//Working Counter: Should remain Zero, If value=1 then data is bad from this device
g_xEP1908_Wc ;

*)

//END_IF ;

END_PROGRAM

// ---- POUs/Control_System_Diagnostics/System_Functions.TcPOU
PROGRAM System_Functions
//		8-2-2012
// 		This Program has been supplied by Beckhoff Automation As-Is and is intended only as an example 
//		implementation. Functionality is not guaranteed. 
//
VAR
	//General timer for periodic reads
	T1									:		TON ;
	xExecute							:		BOOL ;
	tTime1								:		TIME ;

	//Get Device Identification
	fbGetDeviceIdentificationEx			:		FB_GetDeviceIdentificationEx ;
	xGetDeviceId_Busy					:		BOOL ;
	xGetDeviceId_Error					:		BOOL ;
	udiGetDeviceId_ErrId				:		UDINT ;
	stDevIdent							:		ST_DeviceIdentificationEx ;

	//Get ADS Router Info
	fbGetRouterStatusInfo				:		FB_GetRouterStatusInfo ;
	xGetRouterStatusInfo_Busy			:		BOOL ;
	xGetRouterStatusInfo_Error			:		BOOL ;
	udiGetRouterStatusInfo_ErrId		:		UDINT ;
	stRouterStatusInfo					:		ST_TcRouterStatusInfo ;


(*
(* Get CPU Usage Info  *)
	fbTC_CpuUsage: TC_CpuUsage;
	bCpuUsage_Busy: BOOL;
	bCpuUsage_Error: BOOL;
	nCpuUsage_ErrId: UDINT;
	nCpuUsage: UDINT;
	nCpuUsage_HMI: UDINT;

(* Get System Latency Values *)
	fbTC_SysLatency: TC_SysLatency;
	bSysLatency_Busy: BOOL;
	bSysLatency_Error: BOOL;
	nSysLatency_ErrId: UDINT;
	nSysLatency_Actual: UDINT;
	nSysLatency_Max: UDINT;
	nSysLatency_Actual_HMI: UDINT;
	nSysLatency_Max_HMI: UDINT;

(* SystemTaskInfoArr[1].cycleTime is in 100ns increments - needed to convert to ms for display*)
	nCycleTime_HMI: LREAL;

(* SystemTaskInfoArr[1].lastExecTime is in 100ns increments - needed to convert to ms for display*)
	nLastExecTime_HMI: LREAL;
	fbGetDeviceIdentificationEx: FB_GetDeviceIdentificationEx;
*)
	fbFB_MDP_ScanModules				: 		FB_MDP_ScanModules;
	eMDP_ModType						: 		E_MDP_ModuleType;
	usiModIdx							: 		USINT;
	xMDP_ScanModules_busy				: 		BOOL;
	xMDP_ScanModules_Error				: 		BOOL;
	udiMDP_ScanModules_ErrID			: 		UDINT;
	bMDP_ScanModules_DynModID			: 		BYTE;
	usiMDP_ScanModules_ModTypCnt		: 		USINT;
	usiMDP_ScanModules_ModCnt			: 		USINT;

	fbFB_MDP_ReadModuleContent 			:		FB_MDP_ReadModuleContent ;
	ST_MDP_Addr 						:		ST_MDP_Addr ;
	dwMB_Buffer							: 		DWORD ;
	xMDP_Motherboard_ReadModContent_Busy: 		BOOL ;
	xMDP_Motherboard_ReadModContent_Error: 		BOOL ;
	udiMDP_Motherboard_ReadModContent_ErrID: 	UDINT ;
	usiMDP_Motherboard_ReadModContent_ErrPOS: 	USINT ;
	arrMDP_Motherboard_StartIdx			: 		ARRAY [0..255] OF UINT ;

	fbFB_MDP_SplitErrorID				: 		FB_MDP_SplitErrorID ;
	eMDP_ErrGroup 						:		E_MDP_ErrGroup ;
	uiMDP_Motherboard_ReadModContent_ErrCODE:	UINT ;

	fbFB_MDP_ReadModuleHeader			: 		FB_MDP_ReadModuleHeader ;
	xMDP_Motherboard_ReadModHeader_Busy	: 		BOOL ;
	xMDP_Motherboard_ReadModHeader_Error: 		BOOL ;
	udiMDP_Motherboard_ReadModHeader_ErrID: 	UDINT ;
	ST_MDP_Motherboard_ReadModHeader 	:		ST_MDP_ModuleHeader ;

	fbFB_MDP_CPU_Read1					: 		FB_MDP_CPU_Read;
	ST_CPUModHdr 						:		ST_MDP_ModuleHeader ;
	ST_CPUModContent 					: 		ST_MDP_CPU ;

	fbFB_MDP_Mainboard_ReadTBL1			: 		FB_MDP_Mainboard_ReadTBL1;
	ST_MainboardModHdrTBL1				:		ST_MDP_ModuleHeader ;
	ST_MainboardModContentTBL1			: 		ST_MDP_MainboardTBL1 ;

	fbFB_MDP_Mainboard_ReadTBL2			: 		FB_MDP_Mainboard_ReadTBL2 ;
	ST_MainboardModHdrTBL2				:		ST_MDP_ModuleHeader ;
	ST_MainboardModContentTBL2			: 		ST_MDP_MainboardTBL2 ;

	fbFB_MDP_Mainboard_ReadTBL3			: 		FB_MDP_Mainboard_ReadTBL3 ;
	ST_MainboardModHdrTBL3				:		ST_MDP_ModuleHeader ;
	ST_MainboardModContentTBL3			: 		ST_MDP_MainboardTBL3 ;

	fbFB_MDP_Mainboard_ReadTBL4			: 		FB_MDP_Mainboard_ReadTBL4 ;
	ST_MainboardModHdrTBL4				:		ST_MDP_ModuleHeader ;
	ST_MainboardModContentTBL4			: 		ST_MDP_MainboardTBL4 ;
	
	fbFB_MDP_NIC0_Read					: 		FB_MDP_NIC_Read ;
	ST_NIC0_ModHdr						: 		ST_MDP_ModuleHeader ;
	ST_NIC0_ModContent					: 		ST_MDP_NIC_Properties ;
	
	fbFB_MDP_NIC1_Read					: 		FB_MDP_NIC_Read ;
	ST_NIC1_ModHdr						: 		ST_MDP_ModuleHeader ;
	ST_NIC1_ModContent					: 		ST_MDP_NIC_Properties ;	
	lrOperTimeHrs						: 		LREAL ;
	lrOperTimeDays						: 		LREAL ;
	lrOperTimeYears						: 		LREAL ;

	fbFB_MDP_Time1_Read					: 		FB_MDP_Time_ReadTBL1 ;
	ST_Time1_ModHdr						: 		ST_MDP_ModuleHeader ;
	ST_Time1_ModContent					: 		ST_MDP_TimeTBL1 ;

	fbFB_MDP_Time2_Read					: 		FB_MDP_Time_ReadTBL2 ;
	ST_Time2_ModHdr						: 		ST_MDP_ModuleHeader ;
	ST_Time2_ModContent					: 		ST_MDP_TimeTBL2 ;
	
	fbFB_MDP_Memory_Read				: 		FB_MDP_Memory_ReadTBL1 ;
	ST_Memory_ModHdr					: 		ST_MDP_ModuleHeader ;
	ST_Memory_ModContent				: 		ST_MDP_MemoryTBL1 ;
	one									:		INT :=1 ;
	
//	fbFB_MDP_Time1_Read					: 		FB_MDP_Time_ReadTBL1 ;
//	ST_Memory_ModHdr					: 		ST_MDP_ModuleHeader ;
//	ST_Memory_ModContent				: 		ST_MDP_TimeTBL1 ;
	
	testword: INT;
	string45: STRING;
	fbFB_MDP_DiskMngmnt_ReadTBL1		: 		FB_MDP_DiskMngmnt_ReadTBL1 ;
	ST_DiskMngmnt_HdrTBL1				: 		ST_MDP_ModuleHeader ;
	ST_DiskMngmntTBL1					: 		ST_MDP_DiskMngmntTBL1 ;
END_VAR

//		8-2-2012
// 		This Program has been supplied by Beckhoff Automation As-Is and is intended only as an example 
//		implementation. Functionality is not guaranteed. 
//
//   ;
;
testword ;


//IF g_bHMI_ScreenBeingDisplayed = 90 THEN
//Create the xExecute bit for continuous timed interval FB calls
T1(IN:= NOT xExecute, PT:= T#2S, Q=> xExecute, ET=>tTime1 );

(* Computer/Controller Device Info - Get CX and TwinCAT version info
   from the resulting structure "stDevIdent" - display only when the 
   function block is not BUSY retrieving the data else the display
   will "blink" because while the FB is BUSY the values go to 0 or
   "blank" text *)
fbGetDeviceIdentificationEx(
							bExecute					:= 		xExecute, 
							tTimeout					:= 		T#2S, 
							sNetId						:= 		'', 
							bBusy						=> 		xGetDeviceId_Busy, 
							bError						=> 		xGetDeviceId_Error, 
							nErrorID					=> 		udiGetDeviceId_ErrId, 
							stDevIdent					=> 		stDevIdent );
							
IF NOT xGetDeviceId_Busy THEN 
							g_stHMI_DevIdent 			:= 		stDevIdent ; 
END_IF ;

g_stHMI_AppInfo 										:= _AppInfo  ;

//ADS Router Status info
fbGetRouterStatusInfo(		
							sNetId						:= 		'',
							bExecute					:= 		xExecute,
							tTimeout					:= 		T#2S,
							bBusy						=> 		xGetRouterStatusInfo_Busy,
							bError						=> 		xGetRouterStatusInfo_Error,
							nErrID						=> 		udiGetRouterStatusInfo_ErrId,
							info						=> 		stRouterStatusInfo );
							
IF NOT xGetRouterStatusInfo_Busy THEN 
							g_stHMI_RouterStatusInfo	:= 		stRouterStatusInfo ; 
END_IF ;

g_stHMI_PlcTaskSystemInfo 								:= 		_TaskInfo[_AppInfo.TaskCnt] ;
g_lrHMI_PlcTaskSystemInfo_CycleTime 					:= 		g_stHMI_PlcTaskSystemInfo.CycleTime / 10.0 ;
g_lrHMI_PlcTaskSystemInfo_LastExecTime 					:= 		g_stHMI_PlcTaskSystemInfo.LastExecTime / 10.0 ;

//In order to be able to query or set an MDP parameter, the Dynamic Module ID of 
//the module in which the parameter is located must be known.
fbFB_MDP_ScanModules(
							bExecute					:= 		xExecute, 
							nModuleType					:= 		eMDP_ModType, 
							iModIdx						:= 		usiModIdx, 
							tTimeout					:= 		T#2S, 
							sAmsNetId					:= 		'', 
							bBusy						=> 		xMDP_ScanModules_busy, 
							bError						=> 		xMDP_ScanModules_Error, 
							nErrID						=> 		udiMDP_ScanModules_ErrID, 
							nDynModuleId				=> 		bMDP_ScanModules_DynModID, 
							iModuleTypeCount			=> 		usiMDP_ScanModules_ModTypCnt, 
							iModuleCount				=> 		usiMDP_ScanModules_ModCnt );

// The function block enables the header of an MDP module to be queried
fbFB_MDP_ReadModuleHeader(
							bExecute					:= 		xExecute, 
							nDynModuleId				:= 		4, 
							tTimeout					:= 		T#2S, 
							sAmsNetId					:= 		'', 
							bBusy						=> 		xMDP_Motherboard_ReadModHeader_Busy, 
							bError						=> 		xMDP_Motherboard_ReadModHeader_Error, 
							nErrID						=> 		udiMDP_Motherboard_ReadModHeader_ErrID, 
							stMDP_ModHeader				=> 		ST_MDP_Motherboard_ReadModHeader);							
							

fbFB_MDP_CPU_Read1(
							xExecute					:= 		xExecute, 
							tTimeout					:= 		T#2S, 
							usiModIdx					:= 		0, 
							sAmsNetId					:= 		'', 
							bBusy						=> 		, 
							bError						=> 		, 
							nErrID						=> 		, 
							iErrPos						=> 		, 
							stMDP_ModuleHeader			=> 		ST_CPUModHdr, 
							stMDP_ModuleContent			=> 		ST_CPUModContent);							

g_lrHMI_CPUfrequency 									:=		ST_CPUModContent.udiCPUfrequency / 1000.0	; // CPU Clock Frequency in GHz				
g_iHMI_CPUusage											:=		ST_CPUModContent.uiCPUusage ;  // CPU Usage in percent
g_iHMI_CPUtemperature 									:= 		ST_CPUModContent.iCPUtemp ; // CPU Temperature in DegC	

fbFB_MDP_Mainboard_ReadTBL1(
							xExecute					:= 		xExecute, 
							tTimeout					:= 		T#2S, 
							usiModIdx					:= 		0, 
							sAmsNetId					:= 		'', 
							bBusy						=> 		, 
							bError						=> 		, 
							nErrID						=> 		, 
							iErrPos						=> 		, 
							stMDP_ModuleHeader			=> 		ST_MainboardModHdrTBL1, 
							stMDP_ModuleContent			=> 		ST_MainboardModContentTBL1);


g_sHMI_MainboardType 									:= 		ST_MainboardModContentTBL1.sMainboardType ;
g_sHMI_MainboardSN 										:= 		ST_MainboardModContentTBL1.sMainboardSN ;
g_sHMI_MainboardProdDate								:= 		ST_MainboardModContentTBL1.sMainboardProdDate ;
g_udiHMI_MainboardBootCount								:= 		ST_MainboardModContentTBL1.udiMainboardBootCount ;
lrOperTimeHrs											:= 		ST_MainboardModContentTBL1.udiMainboardOperTime / 60.0 ;
lrOperTimeDays											:= 		lrOperTimeHrs / 24.0 ;
g_udiHMI_MainboardOperTimeDays 							:= 		TRUNC(lrOperTimeDays) ;
g_lrHMI_MainboardOperTimeHrs							:=		24.0 * (lrOperTimeDays - UDINT_TO_LREAL(g_udiHMI_MainboardOperTimeDays)) ;
g_diHMI_MainboardMinTemp								:= 		ST_MainboardModContentTBL1.diMainboardMinTemp ;
g_diHMI_MainboardMaxTemp								:= 		ST_MainboardModContentTBL1.diMainboardMaxTemp ;
g_lrHMI_MainboardMinVolt								:= 		ST_MainboardModContentTBL1.diMainboardMinVolt / 1000.0 ;
g_lrHMI_MainboardMaxVolt								:= 		ST_MainboardModContentTBL1.diMainboardMaxVolt / 1000.0 ;
g_iHMI_MainboardActualTemp								:= 		ST_MainboardModContentTBL1.iMainboardActualTemp ;


fbFB_MDP_Mainboard_ReadTBL2(
							xExecute					:= 		xExecute, 
							tTimeout					:= 		T#2S, 
							usiModIdx						:= 		0, 
							sAmsNetId					:= 		'', 
							bBusy						=> 		, 
							bError						=> 		, 
							nErrID						=> 		, 
							iErrPos						=> 		, 
							stMDP_ModuleHeader			=> 		ST_MainboardModHdrTBL2, 
							stMDP_ModuleContent			=> 		ST_MainboardModContentTBL2);


g_bHMI_MainboardRevision 								:= 		ST_MainboardModContentTBL2.usiMainboardRevision ;
g_bHMI_MainboardBiosMajVers 							:= 		ST_MainboardModContentTBL2.usiMainboardBiosMajVers ;
g_bHMI_MainboardBiosMinVers 							:= 		ST_MainboardModContentTBL2.usiMainboardBiosMinVers ;


fbFB_MDP_Mainboard_ReadTBL3(
							xExecute					:= 		xExecute, 
							tTimeout					:= 		T#2S, 
							usiModIdx						:= 		0, 
							sAmsNetId					:= 		'', 
							bBusy						=> 		, 
							bError						=> 		, 
							nErrID						=> 		, 
							iErrPos						=> 		, 
							stMDP_ModuleHeader			=> 		ST_MainboardModHdrTBL3, 
							stMDP_ModuleContent			=> 		ST_MainboardModContentTBL3);							

g_sHMI_Mainboard1p05v 									:= 		ST_MainboardModContentTBL3.sMainboard1p05v ;
g_sHMI_MainboardVccCore 								:= 		ST_MainboardModContentTBL3.sMainboardVccCore ;
g_sHMI_Mainboard5v 										:= 		ST_MainboardModContentTBL3.sMainboard5v ;
g_sHMI_Mainboard12v 									:= 		ST_MainboardModContentTBL3.sMainboard12v ;
g_sHMI_MainboardVBatt 									:= 		ST_MainboardModContentTBL3.sMainboardVBatt ;
g_sHMI_MainboardPwrCtrlVcc 								:= 		ST_MainboardModContentTBL3.sMainboardPwrCtrlVcc ;
g_sHMI_MainboardCX2100_5v 								:= 		ST_MainboardModContentTBL3.sMainboardCX2100_5v ;
g_sHMI_MainboardCX2100_12v 								:= 		ST_MainboardModContentTBL3.sMainboardCX2100_12v ;
g_sHMI_MainboardCX2100_24v 								:= 		ST_MainboardModContentTBL3.sMainboardCX2100_24v ;

					
fbFB_MDP_Mainboard_ReadTBL4(
							xExecute					:= 		xExecute, 
							tTimeout					:= 		T#2S, 
							usiModIdx						:= 		0, 
							sAmsNetId					:= 		'', 
							bBusy						=> 		, 
							bError						=> 		, 
							nErrID						=> 		, 
							iErrPos						=> 		, 
							stMDP_ModuleHeader			=> 		ST_MainboardModHdrTBL4, 
							stMDP_ModuleContent			=> 		ST_MainboardModContentTBL4);

g_lrHMI_Mainboard1p05v 									:= 		ST_MainboardModContentTBL4.iMainboard1p05v / 1000.0 ;
g_lrHMI_MainboardVccCore 								:= 		ST_MainboardModContentTBL4.iMainboardVccCore / 1000.0 ;
g_lrHMI_Mainboard5v 									:= 		ST_MainboardModContentTBL4.iMainboard5v / 1000.0 ;
g_lrHMI_Mainboard12v 									:= 		ST_MainboardModContentTBL4.iMainboard12v / 1000.0 ;
g_lrHMI_MainboardVBatt 									:= 		ST_MainboardModContentTBL4.iMainboardVBatt / 1000.0 ;
g_lrHMI_MainboardPwrCtrlVcc 							:= 		ST_MainboardModContentTBL4.iMainboardPwrCtrlVcc / 1000.0 ;
g_lrHMI_MainboardCX2100_5v 								:= 		ST_MainboardModContentTBL4.iMainboardCX2100_5v / 1000.0 ;
g_lrHMI_MainboardCX2100_12v 							:= 		ST_MainboardModContentTBL4.iMainboardCX2100_12v / 1000.0 ;
g_lrHMI_MainboardCX2100_24v 							:= 		ST_MainboardModContentTBL4.iMainboardCX2100_24v / 1000.0 ; 


fbFB_MDP_NIC0_Read(
							xExecute					:= 		xExecute, 
							tTimeout					:= 		T#2S, 
							usiModIdx					:= 		0, 
							sAmsNetId					:= 		'', 
							bBusy						=> 		, 
							bError						=> 		, 
							nErrID						=> 		, 
							iErrPos						=> 		, 
							stMDP_ModuleHeader			=> 		ST_NIC0_ModHdr, 
							stMDP_ModuleContent			=> 		ST_NIC0_ModContent);

fbFB_MDP_NIC1_Read(
							xExecute					:= 		xExecute, 
							tTimeout					:= 		T#2S, 
							usiModIdx					:= 		1, 
							sAmsNetId					:= 		'', 
							bBusy						=> 		, 
							bError						=> 		, 
							nErrID						=> 		, 
							iErrPos						=> 		, 
							stMDP_ModuleHeader			=> 		ST_NIC1_ModHdr, 
							stMDP_ModuleContent			=> 		ST_NIC1_ModContent);

fbFB_MDP_Time1_Read(
							xExecute					:= 		xExecute, 
							tTimeout					:= 		T#2S, 
							usiModIdx					:= 		0, 
							sAmsNetId					:= 		'', 
							bBusy						=> 		, 
							bError						=> 		, 
							nErrID						=> 		, 
							iErrPos						=> 		, 
							stMDP_ModuleHeader			=> 		ST_Time1_ModHdr, 
							stMDP_ModuleContent			=> 		ST_Time1_ModContent);				

g_sHMI_SNTP_Server										:= 		ST_Time1_ModContent.sSNTP_Server ;
g_lrHMI_SNTP_Refresh_Minutes							:= 		UDINT_TO_LREAL(ST_Time1_ModContent.udiSNTP_Refresh) / 60.0 ; // Seconds / 60 = Minutes
g_lrHMI_Years_Since_1_1_1970							:= 		UDINT_TO_LREAL(ST_Time1_ModContent.udiSec_Since_1_1_1970) / (60 * 60 *24 * 365) ;
g_sHMI_DateTime_Presentation							:= 		ST_Time1_ModContent.sDateTime_Presentation ;
g_uiHMI_Timezone										:= 		ST_Time1_ModContent.uiTimezone ;


fbFB_MDP_Time2_Read(
							xExecute					:= 		xExecute, 
							tTimeout					:= 		T#2S, 
							usiModIdx					:= 		0, 
							sAmsNetId					:= 		'', 
							bBusy						=> 		, 
							bError						=> 		, 
							nErrID						=> 		, 
							iErrPos						=> 		, 
							stMDP_ModuleHeader			=> 		ST_Time2_ModHdr, 
							stMDP_ModuleContent			=> 		ST_Time2_ModContent);
							
IF ST_Time1_ModContent.uiTimezone = 0 THEN
	g_sHMI_currentTimeZone := ST_Time2_ModContent.sTimezone1 ;
ELSIF ST_Time1_ModContent.uiTimezone = 1 THEN
	g_sHMI_currentTimeZone := ST_Time2_ModContent.sTimezone2 ;
ELSIF ST_Time1_ModContent.uiTimezone = 2 THEN
	g_sHMI_currentTimeZone := ST_Time2_ModContent.sTimezone3 ;
ELSIF ST_Time1_ModContent.uiTimezone = 3 THEN
	g_sHMI_currentTimeZone := ST_Time2_ModContent.sTimezone4 ;
ELSIF ST_Time1_ModContent.uiTimezone = 4 THEN
	g_sHMI_currentTimeZone := ST_Time2_ModContent.sTimezone5 ;	
ELSIF ST_Time1_ModContent.uiTimezone = 5 THEN
	g_sHMI_currentTimeZone := ST_Time2_ModContent.sTimezone6 ;
ELSIF ST_Time1_ModContent.uiTimezone = 6 THEN
	g_sHMI_currentTimeZone := ST_Time2_ModContent.sTimezone7 ;
ELSIF ST_Time1_ModContent.uiTimezone = 7 THEN
	g_sHMI_currentTimeZone := ST_Time2_ModContent.sTimezone8 ;
ELSIF ST_Time1_ModContent.uiTimezone = 8 THEN
	g_sHMI_currentTimeZone := ST_Time2_ModContent.sTimezone9 ;		
ELSIF ST_Time1_ModContent.uiTimezone = 9 THEN
	g_sHMI_currentTimeZone := ST_Time2_ModContent.sTimezone10 ;
ELSIF ST_Time1_ModContent.uiTimezone = 10 THEN
	g_sHMI_currentTimeZone := ST_Time2_ModContent.sTimezone11 ;
ELSIF ST_Time1_ModContent.uiTimezone = 11 THEN
	g_sHMI_currentTimeZone := ST_Time2_ModContent.sTimezone12 ;
ELSIF ST_Time1_ModContent.uiTimezone = 12 THEN
	g_sHMI_currentTimeZone := ST_Time2_ModContent.sTimezone13 ;	
ELSIF ST_Time1_ModContent.uiTimezone = 13 THEN
	g_sHMI_currentTimeZone := ST_Time2_ModContent.sTimezone14 ;
ELSIF ST_Time1_ModContent.uiTimezone = 14 THEN
	g_sHMI_currentTimeZone := ST_Time2_ModContent.sTimezone15 ;
ELSIF ST_Time1_ModContent.uiTimezone = 15 THEN
	g_sHMI_currentTimeZone := ST_Time2_ModContent.sTimezone16 ;
ELSIF ST_Time1_ModContent.uiTimezone = 16 THEN
	g_sHMI_currentTimeZone := ST_Time2_ModContent.sTimezone17 ;		
ELSIF ST_Time1_ModContent.uiTimezone = 17 THEN
	g_sHMI_currentTimeZone := ST_Time2_ModContent.sTimezone18 ;
ELSIF ST_Time1_ModContent.uiTimezone = 18 THEN
	g_sHMI_currentTimeZone := ST_Time2_ModContent.sTimezone19 ;
ELSIF ST_Time1_ModContent.uiTimezone = 19 THEN
	g_sHMI_currentTimeZone := ST_Time2_ModContent.sTimezone20 ;
ELSIF ST_Time1_ModContent.uiTimezone = 20 THEN
	g_sHMI_currentTimeZone := ST_Time2_ModContent.sTimezone21 ;	
ELSIF ST_Time1_ModContent.uiTimezone = 21 THEN
	g_sHMI_currentTimeZone := ST_Time2_ModContent.sTimezone22 ;
ELSIF ST_Time1_ModContent.uiTimezone = 22 THEN
	g_sHMI_currentTimeZone := ST_Time2_ModContent.sTimezone23 ;
ELSIF ST_Time1_ModContent.uiTimezone = 23 THEN
	g_sHMI_currentTimeZone := ST_Time2_ModContent.sTimezone24 ;
ELSIF ST_Time1_ModContent.uiTimezone = 24 THEN
	g_sHMI_currentTimeZone := ST_Time2_ModContent.sTimezone25 ;		
ELSIF ST_Time1_ModContent.uiTimezone = 25 THEN
	g_sHMI_currentTimeZone := ST_Time2_ModContent.sTimezone26 ;
ELSIF ST_Time1_ModContent.uiTimezone = 26 THEN
	g_sHMI_currentTimeZone := ST_Time2_ModContent.sTimezone27 ;
ELSIF ST_Time1_ModContent.uiTimezone = 27 THEN
	g_sHMI_currentTimeZone := ST_Time2_ModContent.sTimezone28 ;
ELSIF ST_Time1_ModContent.uiTimezone = 28 THEN
	g_sHMI_currentTimeZone := ST_Time2_ModContent.sTimezone29 ;	
ELSIF ST_Time1_ModContent.uiTimezone = 29 THEN
	g_sHMI_currentTimeZone := ST_Time2_ModContent.sTimezone30 ;
ELSIF ST_Time1_ModContent.uiTimezone = 30 THEN
	g_sHMI_currentTimeZone := ST_Time2_ModContent.sTimezone31 ;
ELSIF ST_Time1_ModContent.uiTimezone = 31 THEN
	g_sHMI_currentTimeZone := ST_Time2_ModContent.sTimezone32 ;
ELSIF ST_Time1_ModContent.uiTimezone = 32 THEN
	g_sHMI_currentTimeZone := ST_Time2_ModContent.sTimezone33 ;			
ELSIF ST_Time1_ModContent.uiTimezone = 33 THEN
	g_sHMI_currentTimeZone := ST_Time2_ModContent.sTimezone34 ;
ELSIF ST_Time1_ModContent.uiTimezone = 34 THEN
	g_sHMI_currentTimeZone := ST_Time2_ModContent.sTimezone35 ;
ELSIF ST_Time1_ModContent.uiTimezone = 35 THEN
	g_sHMI_currentTimeZone := ST_Time2_ModContent.sTimezone36 ;
ELSIF ST_Time1_ModContent.uiTimezone = 36 THEN
	g_sHMI_currentTimeZone := ST_Time2_ModContent.sTimezone37 ;	
ELSIF ST_Time1_ModContent.uiTimezone = 37 THEN
	g_sHMI_currentTimeZone := ST_Time2_ModContent.sTimezone38 ;
ELSIF ST_Time1_ModContent.uiTimezone = 38 THEN
	g_sHMI_currentTimeZone := ST_Time2_ModContent.sTimezone39 ;
ELSIF ST_Time1_ModContent.uiTimezone = 39 THEN
	g_sHMI_currentTimeZone := ST_Time2_ModContent.sTimezone40 ;
ELSIF ST_Time1_ModContent.uiTimezone = 40 THEN
	g_sHMI_currentTimeZone := ST_Time2_ModContent.sTimezone41 ;		
ELSIF ST_Time1_ModContent.uiTimezone = 41 THEN
	g_sHMI_currentTimeZone := ST_Time2_ModContent.sTimezone42 ;
ELSIF ST_Time1_ModContent.uiTimezone = 42 THEN
	g_sHMI_currentTimeZone := ST_Time2_ModContent.sTimezone43 ;
ELSIF ST_Time1_ModContent.uiTimezone = 43 THEN
	g_sHMI_currentTimeZone := ST_Time2_ModContent.sTimezone44 ;
ELSIF ST_Time1_ModContent.uiTimezone = 44 THEN
	g_sHMI_currentTimeZone := ST_Time2_ModContent.sTimezone45 ;	
ELSIF ST_Time1_ModContent.uiTimezone = 45 THEN
	g_sHMI_currentTimeZone := ST_Time2_ModContent.sTimezone46 ;
ELSIF ST_Time1_ModContent.uiTimezone = 46 THEN
	g_sHMI_currentTimeZone := ST_Time2_ModContent.sTimezone47 ;
ELSIF ST_Time1_ModContent.uiTimezone = 47 THEN
	g_sHMI_currentTimeZone := ST_Time2_ModContent.sTimezone48 ;
ELSIF ST_Time1_ModContent.uiTimezone = 48 THEN
	g_sHMI_currentTimeZone := ST_Time2_ModContent.sTimezone49 ;		
ELSIF ST_Time1_ModContent.uiTimezone = 49 THEN
	g_sHMI_currentTimeZone := ST_Time2_ModContent.sTimezone50 ;
ELSIF ST_Time1_ModContent.uiTimezone = 50 THEN
	g_sHMI_currentTimeZone := ST_Time2_ModContent.sTimezone51 ;
ELSIF ST_Time1_ModContent.uiTimezone = 51 THEN
	g_sHMI_currentTimeZone := ST_Time2_ModContent.sTimezone52 ;
ELSIF ST_Time1_ModContent.uiTimezone = 52 THEN
	g_sHMI_currentTimeZone := ST_Time2_ModContent.sTimezone53 ;	
ELSIF ST_Time1_ModContent.uiTimezone = 53 THEN
	g_sHMI_currentTimeZone := ST_Time2_ModContent.sTimezone54 ;
ELSIF ST_Time1_ModContent.uiTimezone = 54 THEN
	g_sHMI_currentTimeZone := ST_Time2_ModContent.sTimezone55 ;
ELSIF ST_Time1_ModContent.uiTimezone = 55 THEN
	g_sHMI_currentTimeZone := ST_Time2_ModContent.sTimezone56 ;
ELSIF ST_Time1_ModContent.uiTimezone = 56 THEN
	g_sHMI_currentTimeZone := ST_Time2_ModContent.sTimezone57 ;		
ELSIF ST_Time1_ModContent.uiTimezone = 57 THEN
	g_sHMI_currentTimeZone := ST_Time2_ModContent.sTimezone58 ;
ELSIF ST_Time1_ModContent.uiTimezone = 58 THEN
	g_sHMI_currentTimeZone := ST_Time2_ModContent.sTimezone59 ;
ELSIF ST_Time1_ModContent.uiTimezone = 59 THEN
	g_sHMI_currentTimeZone := ST_Time2_ModContent.sTimezone60 ;
ELSIF ST_Time1_ModContent.uiTimezone = 60 THEN
	g_sHMI_currentTimeZone := ST_Time2_ModContent.sTimezone61 ;	
ELSIF ST_Time1_ModContent.uiTimezone = 61 THEN
	g_sHMI_currentTimeZone := ST_Time2_ModContent.sTimezone62 ;
ELSIF ST_Time1_ModContent.uiTimezone = 62 THEN
	g_sHMI_currentTimeZone := ST_Time2_ModContent.sTimezone63 ;
ELSIF ST_Time1_ModContent.uiTimezone = 63 THEN
	g_sHMI_currentTimeZone := ST_Time2_ModContent.sTimezone64 ;
ELSIF ST_Time1_ModContent.uiTimezone = 64 THEN
	g_sHMI_currentTimeZone := ST_Time2_ModContent.sTimezone65 ;	
ELSIF ST_Time1_ModContent.uiTimezone = 65 THEN
	g_sHMI_currentTimeZone := ST_Time2_ModContent.sTimezone66 ;
ELSIF ST_Time1_ModContent.uiTimezone = 66 THEN
	g_sHMI_currentTimeZone := ST_Time2_ModContent.sTimezone67 ;
ELSIF ST_Time1_ModContent.uiTimezone = 67 THEN
	g_sHMI_currentTimeZone := ST_Time2_ModContent.sTimezone68 ;
ELSIF ST_Time1_ModContent.uiTimezone = 68 THEN
	g_sHMI_currentTimeZone := ST_Time2_ModContent.sTimezone69 ;	
ELSIF ST_Time1_ModContent.uiTimezone = 69 THEN
	g_sHMI_currentTimeZone := ST_Time2_ModContent.sTimezone70 ;
ELSIF ST_Time1_ModContent.uiTimezone = 70 THEN
	g_sHMI_currentTimeZone := ST_Time2_ModContent.sTimezone71 ;
ELSIF ST_Time1_ModContent.uiTimezone = 71 THEN
	g_sHMI_currentTimeZone := ST_Time2_ModContent.sTimezone72 ;
ELSIF ST_Time1_ModContent.uiTimezone = 72 THEN
	g_sHMI_currentTimeZone := ST_Time2_ModContent.sTimezone73 ;		
ELSIF ST_Time1_ModContent.uiTimezone = 73 THEN
	g_sHMI_currentTimeZone := ST_Time2_ModContent.sTimezone74 ;
ELSIF ST_Time1_ModContent.uiTimezone = 74 THEN
	g_sHMI_currentTimeZone := ST_Time2_ModContent.sTimezone75 ;
ELSIF ST_Time1_ModContent.uiTimezone = 75 THEN
	g_sHMI_currentTimeZone := ST_Time2_ModContent.sTimezone76 ;
ELSIF ST_Time1_ModContent.uiTimezone = 76 THEN
	g_sHMI_currentTimeZone := ST_Time2_ModContent.sTimezone77 ;	
ELSIF ST_Time1_ModContent.uiTimezone = 77 THEN
	g_sHMI_currentTimeZone := ST_Time2_ModContent.sTimezone78 ;
ELSIF ST_Time1_ModContent.uiTimezone = 78 THEN
	g_sHMI_currentTimeZone := ST_Time2_ModContent.sTimezone79 ;
ELSIF ST_Time1_ModContent.uiTimezone = 79 THEN
	g_sHMI_currentTimeZone := ST_Time2_ModContent.sTimezone80 ;
ELSIF ST_Time1_ModContent.uiTimezone = 80 THEN
	g_sHMI_currentTimeZone := ST_Time2_ModContent.sTimezone81 ;		
ELSIF ST_Time1_ModContent.uiTimezone = 81 THEN
	g_sHMI_currentTimeZone := ST_Time2_ModContent.sTimezone82 ;
ELSIF ST_Time1_ModContent.uiTimezone = 82 THEN
	g_sHMI_currentTimeZone := ST_Time2_ModContent.sTimezone83 ;
ELSIF ST_Time1_ModContent.uiTimezone = 83 THEN
	g_sHMI_currentTimeZone := ST_Time2_ModContent.sTimezone84 ;
ELSIF ST_Time1_ModContent.uiTimezone = 84 THEN
	g_sHMI_currentTimeZone := ST_Time2_ModContent.sTimezone85 ;	
ELSIF ST_Time1_ModContent.uiTimezone = 85 THEN
	g_sHMI_currentTimeZone := ST_Time2_ModContent.sTimezone86 ;
ELSIF ST_Time1_ModContent.uiTimezone = 86 THEN
	g_sHMI_currentTimeZone := ST_Time2_ModContent.sTimezone87 ;
ELSIF ST_Time1_ModContent.uiTimezone = 87 THEN
	g_sHMI_currentTimeZone := ST_Time2_ModContent.sTimezone88 ;
ELSIF ST_Time1_ModContent.uiTimezone = 88 THEN
	g_sHMI_currentTimeZone := ST_Time2_ModContent.sTimezone89 ;		
ELSIF ST_Time1_ModContent.uiTimezone = 89 THEN
	g_sHMI_currentTimeZone := ST_Time2_ModContent.sTimezone90 ;
ELSIF ST_Time1_ModContent.uiTimezone = 90 THEN
	g_sHMI_currentTimeZone := ST_Time2_ModContent.sTimezone91 ;
ELSIF ST_Time1_ModContent.uiTimezone = 91 THEN
	g_sHMI_currentTimeZone := ST_Time2_ModContent.sTimezone92 ;
ELSIF ST_Time1_ModContent.uiTimezone = 92 THEN
	g_sHMI_currentTimeZone := ST_Time2_ModContent.sTimezone93 ;	
ELSIF ST_Time1_ModContent.uiTimezone = 93 THEN
	g_sHMI_currentTimeZone := ST_Time2_ModContent.sTimezone94 ;
ELSIF ST_Time1_ModContent.uiTimezone = 94 THEN
	g_sHMI_currentTimeZone := ST_Time2_ModContent.sTimezone95 ;
ELSIF ST_Time1_ModContent.uiTimezone = 95 THEN
	g_sHMI_currentTimeZone := ST_Time2_ModContent.sTimezone96 ;
ELSIF ST_Time1_ModContent.uiTimezone = 96 THEN
	g_sHMI_currentTimeZone := ST_Time2_ModContent.sTimezone97 ;			
ELSIF ST_Time1_ModContent.uiTimezone = 97 THEN
	g_sHMI_currentTimeZone := ST_Time2_ModContent.sTimezone98 ;
ELSIF ST_Time1_ModContent.uiTimezone = 98 THEN
	g_sHMI_currentTimeZone := ST_Time2_ModContent.sTimezone99 ;
ELSIF ST_Time1_ModContent.uiTimezone = 99 THEN
	g_sHMI_currentTimeZone := ST_Time2_ModContent.sTimezone100 ;
ELSIF ST_Time1_ModContent.uiTimezone = 100 THEN
	g_sHMI_currentTimeZone := ST_Time2_ModContent.sTimezone101 ;	
END_IF
							
fbFB_MDP_Memory_Read(
							xExecute					:= 		xExecute, 
							tTimeout					:= 		T#2S, 
							usiModIdx					:= 		0, 
							sAmsNetId					:= 		'', 
							bBusy						=> 		, 
							bError						=> 		, 
							nErrID						=> 		, 
							iErrPos						=> 		, 
							stMDP_ModuleHeader			=> 		ST_Memory_ModHdr, 
							stMDP_ModuleContent			=> 		ST_Memory_ModContent);		

	g_lrHMI_ProgMemAllocated_InGB 		:= UDINT_TO_LREAL(ST_Memory_ModContent.udiProgMemAllocated) / 1000000000.0 ;	
	g_lrHMI_ProgMemAvailable_InGB 		:= UDINT_TO_LREAL(ST_Memory_ModContent.udiProgMemAvailable) / 1000000000.0 ;	
	g_lrHMI_ProgMemUsed_InGB 			:= g_lrHMI_ProgMemAllocated_InGB - g_lrHMI_ProgMemAvailable_InGB ;	
	g_lrHMI_ProgStorAllocated_InGB 		:= UDINT_TO_LREAL(ST_Memory_ModContent.udiStorageMemAllocated) / 1000000000.0 ;	
	g_lrHMI_ProgStorAvailable_InGB 		:= UDINT_TO_LREAL(ST_Memory_ModContent.udiStorageMemAvailable) / 1000000000.0 ;	
	g_lrHMI_ProgStorUsed_InGB 			:= g_lrHMI_ProgStorAllocated_InGB - g_lrHMI_ProgStorAvailable_InGB ;
	g_lrHMI_ProgStorMemDivision_InGB	:= UDINT_TO_LREAL(ST_Memory_ModContent.udiMemoryDivision) / 1000000000.0 ;	


fbFB_MDP_DiskMngmnt_ReadTBL1(
								xExecute				:= 		xExecute, 
								tTimeout				:= 		T#2S, 
								usiModIdx				:= 		0, 
								sAmsNetId				:= 		'', 
								bBusy					=> 		, 
								bError					=> 		, 
								nErrID					=> 		, 
								iErrPos					=> 		, 
								stMDP_ModuleHeader		=> 		ST_DiskMngmnt_HdrTBL1, 
								stMDP_ModuleContent		=> 		ST_DiskMngmntTBL1);








							
fbFB_MDP_Time1_Read(
							xExecute					:= 		xExecute, 
							tTimeout					:= 		T#2S, 
							usiModIdx					:= 		0, 
							sAmsNetId					:= 		'', 
							bBusy						=> 		, 
							bError						=> 		, 
							nErrID						=> 		, 
							iErrPos						=> 		, 
							stMDP_ModuleHeader			=> 		ST_Time1_ModHdr, 
							stMDP_ModuleContent			=> 		ST_Time1_ModContent);					
//	END_IF ;

END_PROGRAM

// ---- POUs/MDP_Function_Blocks/FB_MDP_CPU_Read.TcPOU
FUNCTION_BLOCK FB_MDP_CPU_Read

VAR_INPUT
	xExecute			: BOOL;								// Function block execution is triggered by a rising edge at this input
	tTimeout			: TIME		:= DEFAULT_ADS_TIMEOUT;	// States the time before the function is cancelled
	usiModIdx			: USINT		:= 0;					// Index number of chosen MDP device
	sAmsNetId			: T_AmsNetId;						// keep empty '' for the local device
END_VAR

VAR_OUTPUT
	xBusy				: BOOL;
	xError				: BOOL;
	udiErrID			: UDINT;
	usiErrPos			: USINT;							//If a subindex is not supported, iErrPos indicates at which subindex the error appears first
	stMDP_ModuleHeader	: ST_MDP_ModuleHeader;
	stMDP_ModuleContent	: ST_MDP_CPU;	
END_VAR

VAR
	fbMDP_ReadModule: FB_MDP_ReadModule;
	arrData				: ARRAY[0..15] OF BYTE;				// requested data
	arrStartIdx			: ARRAY[0..255] OF UINT;			// startindexes in bytes of each subindex element

	stMDP_Addr			: ST_MDP_Addr;
	eModuleType			: E_MDP_ModuleType;
	usiSubIdxCount		: USINT;

	xSubExecute			: BOOL;
	xReadBusy			: BOOL;

	RisingEdge			: R_TRIG;
	TimeOut				: TON;								// general timeout	
END_VAR

RisingEdge( CLK					:= xExecute );
IF NOT xBusy THEN											// FB only react to the external execute if it is not busy
	IF RisingEdge.Q THEN
		xBusy					:= TRUE;

		// reset variables
		xError					:= FALSE;
		udiErrID				:= 0;
		usiErrPos				:= 0;
		xSubExecute				:= TRUE;

		// specific values for CPU content
		stMDP_Addr.nArea		:= 16#08;
//		stMDP_Addr.nModuleId;								will be allocated dynamically
		stMDP_Addr.nTableId		:= 16#01;
//		stMDP_Addr.nFlag;									not used at ths time
//		stMDP_Addr.nSubIdx;									all subindexes will be requested
		eModuleType				:= eMDP_ModT_CPU;
		usiSubIdxCount			:= 4;						// TableId 16#01 contains 3 elements

		MEMSET( ADR(arrData), 0, SIZEOF(arrData) );			// reset buffer

		TimeOut(IN 				:= FALSE);
		TimeOut(PT 				:= tTimeout, IN 	:= TRUE);
	END_IF
END_IF


IF xBusy THEN
	IF xSubExecute THEN
		xSubExecute 			:= FALSE;

		fbMDP_ReadModule( bExecute := FALSE );
		fbMDP_ReadModule(
			stMDP_Addr			:= stMDP_Addr,
			eModuleType			:= eModuleType,
			iModIdx				:= usiModIdx,
			iSubIdxCount		:= usiSubIdxCount,
			bExecute			:= TRUE,
			tTimeout			:= tTimeout,
			pDstBuf				:= ADR(arrData),
			cbDstBufLen			:= SIZEOF(arrData),
			sAmsNetId			:= sAmsNetId,

			bBusy				=> xReadBusy,
			bError				=> xError,
			nErrID				=> udiErrID,
			iErrPos				=> usiErrPos,
			stMDP_DynAddr		=> ,
			iModuleTypeCount	=> ,
			iModuleCount		=> ,
			stMDP_ModuleHeader	=> ,
			arrStartIdx			=> ,
		);
	ELSE
		fbMDP_ReadModule(
			bExecute			:= FALSE,

			bBusy				=> xReadBusy,
			bError				=> xError,
			nErrID 				=> udiErrID,
			iErrPos				=> usiErrPos,
		 );
		IF NOT xReadBusy THEN
			// allocate received module header
			stMDP_ModuleHeader	:= fbMDP_ReadModule.stMDP_ModuleHeader;
			// allocate information of startindexes in data buffer
			MEMCPY(ADR(arrStartIdx), ADR(fbMDP_ReadModule.arrStartIdx), SIZEOF(arrStartIdx) );
			// reset module content struct
			MEMSET( ADR(stMDP_ModuleContent), 0, SIZEOF(stMDP_ModuleContent) );
			// allocate received data to NIC struct
			stMDP_ModuleContent.uiLen		:= arrData[0];
			MEMCPY(ADR(stMDP_ModuleContent.udiCPUfrequency), 	ADR(arrData)+arrStartIdx[1], MIN(arrStartIdx[2]-arrStartIdx[1], SIZEOF(stMDP_ModuleContent.udiCPUfrequency)) );
			MEMCPY(ADR(stMDP_ModuleContent.uiCPUusage), 		ADR(arrData)+arrStartIdx[2], MIN(arrStartIdx[3]-arrStartIdx[2], SIZEOF(stMDP_ModuleContent.uiCPUusage))     );
			MEMCPY(ADR(stMDP_ModuleContent.iCPUtemp), 			ADR(arrData)+arrStartIdx[3], MIN(arrStartIdx[4]-arrStartIdx[3], SIZEOF(stMDP_ModuleContent.iCPUtemp))     );

			// reset FB
			xBusy 				:= FALSE;
		END_IF
	END_IF

	
	// check timeout
	TimeOut();
	IF TimeOut.Q THEN
		TimeOut(IN 				:= FALSE);
		xError					:= TRUE;
		udiErrID				:= INT_TO_UINT(eMDP_Err_PLC) * 16#10000 + INT_TO_UINT(eMDP_ErrPLC_TimeOut);
	END_IF
END_IF

IF xError THEN
	// reset FB
	xBusy := FALSE;
END_IF

END_FUNCTION_BLOCK

// ---- POUs/MDP_Function_Blocks/FB_MDP_Mainboard_ReadTBL2.TcPOU
FUNCTION_BLOCK FB_MDP_Mainboard_ReadTBL2

VAR_INPUT
	xExecute			: BOOL;								// Function block execution is triggered by a rising edge at this input
	tTimeout			: TIME		:= DEFAULT_ADS_TIMEOUT;	// States the time before the function is cancelled
	usiModIdx			: USINT		:= 0;					// Index number of chosen MDP device 
	sAmsNetId			: T_AmsNetId;						// keep empty '' for the local device
END_VAR

VAR_OUTPUT
	xBusy				: BOOL;
	xError				: BOOL;
	udiErrID			: UDINT;
	usiErrPos			: USINT;							// If a subindex is not supported, iErrPos indicates at which subindex the error appears first
	stMDP_ModuleHeader	: ST_MDP_ModuleHeader;
	stMDP_ModuleContent	: ST_MDP_MainboardTBL2;	
END_VAR

VAR
	fbMDP_ReadModule: FB_MDP_ReadModule;
	arrData				: ARRAY[0..5] OF BYTE;				// requested data
	arrStartIdx			: ARRAY[0..4] OF UINT;				// startindexes in bytes of each subindex element

	stMDP_Addr			: ST_MDP_Addr;
	eModuleType			: E_MDP_ModuleType;
	usiSubIdxCount		: USINT;

	xSubExecute			: BOOL;
	xReadBusy			: BOOL;

	RisingEdge			: R_TRIG;
	TimeOut				: TON;								// general timeout	
END_VAR

RisingEdge( CLK					:= xExecute );
IF NOT xBusy THEN										// FB only react to the external execute if it is not busy
	IF RisingEdge.Q THEN
		xBusy					:= TRUE;
		// reset variables
		xError					:= FALSE;
		udiErrID				:= 0;
		usiErrPos				:= 0;
		xSubExecute				:= TRUE;

		// specific values for Mainboard content
		stMDP_Addr.nArea		:= 16#08;
//		stMDP_Addr.nModuleId;							will be allocated dynamically
		stMDP_Addr.nTableId		:= 16#02;
//		stMDP_Addr.nFlag;								not used up to now
//		stMDP_Addr.nSubIdx;								all subindexes will be requested
		eModuleType				:= eMDP_ModT_Mainboard;
		usiSubIdxCount			:= 4;					// TableId 16#01 contains 3 elements

		MEMSET( ADR(arrData), 0, SIZEOF(arrData) );		// reset buffer

		TimeOut(IN 				:= FALSE);
		TimeOut(PT 				:= tTimeout, IN 	:= TRUE);
	END_IF
END_IF


IF xBusy THEN
	IF xSubExecute THEN
		xSubExecute 			:= FALSE;

		fbMDP_ReadModule( bExecute := FALSE );
		fbMDP_ReadModule(
			stMDP_Addr			:= stMDP_Addr,
			eModuleType			:= eModuleType,
			iModIdx				:= usiModIdx,
			iSubIdxCount		:= usiSubIdxCount,
			bExecute			:= TRUE,
			tTimeout			:= tTimeout,
			pDstBuf				:= ADR(arrData),
			cbDstBufLen			:= SIZEOF(arrData),
			sAmsNetId			:= sAmsNetId,

			bBusy				=> xReadBusy,
			bError				=> xError,
			nErrID				=> udiErrID,
			iErrPos				=> usiErrPos,
			stMDP_DynAddr		=> ,
			iModuleTypeCount	=> ,
			iModuleCount		=> ,
			stMDP_ModuleHeader	=> ,
			arrStartIdx			=> ,
		);
	ELSE
		fbMDP_ReadModule(
			bExecute			:= FALSE,

			bBusy				=> xReadBusy,
			bError				=> xError,
			nErrID 				=> udiErrID,
			iErrPos				=> usiErrPos,
		 );
		IF NOT xReadBusy THEN
			// allocate received module header
			stMDP_ModuleHeader	:= fbMDP_ReadModule.stMDP_ModuleHeader;
			// allocate information of startindexes in data buffer
			MEMCPY(ADR(arrStartIdx), ADR(fbMDP_ReadModule.arrStartIdx), SIZEOF(arrStartIdx) );
			// reset module content struct
			MEMSET( ADR(stMDP_ModuleContent), 0, SIZEOF(stMDP_ModuleContent) );
			// allocate received data to NIC struct
			stMDP_ModuleContent.uiLen		:= arrData[0];
			MEMCPY(ADR(stMDP_ModuleContent.usiMainboardRevision),			ADR(arrData)+arrStartIdx[1],	MIN(arrStartIdx[2]-arrStartIdx[1],	SIZEOF(stMDP_ModuleContent.usiMainboardRevision))     );
			MEMCPY(ADR(stMDP_ModuleContent.usiMainboardBiosMajVers),		ADR(arrData)+arrStartIdx[2],	MIN(arrStartIdx[3]-arrStartIdx[2],	SIZEOF(stMDP_ModuleContent.usiMainboardBiosMajVers))     );
			MEMCPY(ADR(stMDP_ModuleContent.usiMainboardBiosMinVers),		ADR(arrData)+arrStartIdx[3],	MIN(arrStartIdx[4]-arrStartIdx[3],	SIZEOF(stMDP_ModuleContent.usiMainboardBiosMinVers))     );

			// reset FB
			xBusy 				:= FALSE;
		END_IF
	END_IF

	// check timeout
	TimeOut();
	IF TimeOut.Q THEN
		TimeOut(IN 				:= FALSE);
		xError					:= TRUE;
		udiErrID				:= INT_TO_UINT(eMDP_Err_PLC) * 16#10000 + INT_TO_UINT(eMDP_ErrPLC_TimeOut);
	END_IF
END_IF

IF xError THEN
	// reset FB
	xBusy 						:= FALSE;
END_IF

END_FUNCTION_BLOCK

// ---- POUs/MDP_Function_Blocks/FB_MDP_Mainboard_ReadTBL3.TcPOU
FUNCTION_BLOCK FB_MDP_Mainboard_ReadTBL3

VAR_INPUT
	xExecute				: BOOL;								// Function block execution is triggered by a rising edge at this input
	tTimeout				: TIME		:= DEFAULT_ADS_TIMEOUT;	// States the time before the function is cancelled
	usiModIdx				: USINT		:= 0;					// Index number of chosen MDP device
	sAmsNetId				: T_AmsNetId;						// keep empty '' for the local device
END_VAR

VAR_OUTPUT
	xBusy					: BOOL;
	xError					: BOOL;
	udiErrID				: UDINT;
	usiErrPos				: USINT;							// If a subindex is not supported, iErrPos indicates at which subindex the error appears first
	stMDP_ModuleHeader		: ST_MDP_ModuleHeader;
	stMDP_ModuleContent		: ST_MDP_MainboardTBL3;	
END_VAR

VAR
	fbMDP_ReadModule		: FB_MDP_ReadModule;
	arrData					: ARRAY[0..70] OF BYTE;				// requested data
	arrStartIdx				: ARRAY[0..11] OF UINT;				// startindexes in bytes of each subindex element

	stMDP_Addr				: ST_MDP_Addr;
	eModuleType				: E_MDP_ModuleType;
	usiSubIdxCount			: USINT;

	xSubExecute				: BOOL;
	xReadBusy				: BOOL;

	RisingEdge				: R_TRIG;
	TimeOut					: TON;								// general timeout	
END_VAR

RisingEdge( CLK					:= xExecute );
IF NOT xBusy THEN											// FB only react to the external execute if it is not busy
	IF RisingEdge.Q THEN
		xBusy					:= TRUE;

		// reset variables
		xError					:= FALSE;
		udiErrID				:= 0;
		usiErrPos				:= 0;
		xSubExecute				:= TRUE;

		// specific values for Mainboard content
		stMDP_Addr.nArea		:= 16#08;
//		stMDP_Addr.nModuleId;								will be allocated dynamically
		stMDP_Addr.nTableId		:= 16#03;
//		stMDP_Addr.nFlag;									not used at this time
//		stMDP_Addr.nSubIdx;									all subindexes will be requested
		eModuleType				:= eMDP_ModT_Mainboard;
		usiSubIdxCount			:= 10;						// TableId 16#01 contains 9 elements

		MEMSET( ADR(arrData), 0, SIZEOF(arrData) );			// reset buffer

		TimeOut(IN 				:= FALSE);
		TimeOut(PT 				:= tTimeout, IN 	:= TRUE);
	END_IF
END_IF


IF xBusy THEN
	IF xSubExecute THEN
		xSubExecute 			:= FALSE;

		fbMDP_ReadModule( bExecute := FALSE );
		fbMDP_ReadModule(
			stMDP_Addr			:= stMDP_Addr,
			eModuleType			:= eModuleType,
			iModIdx				:= usiModIdx,
			iSubIdxCount		:= usiSubIdxCount,
			bExecute			:= TRUE,
			tTimeout			:= tTimeout,
			pDstBuf				:= ADR(arrData),
			cbDstBufLen			:= SIZEOF(arrData),
			sAmsNetId			:= sAmsNetId,

			bBusy				=> xReadBusy,
			bError				=> xError,
			nErrID				=> udiErrID,
			iErrPos				=> usiErrPos,
			stMDP_DynAddr		=> ,
			iModuleTypeCount	=> ,
			iModuleCount		=> ,
			stMDP_ModuleHeader	=> ,
			arrStartIdx			=> ,
		);
	ELSE
		fbMDP_ReadModule(
			bExecute			:= FALSE,

			bBusy				=> xReadBusy,
			bError				=> xError,
			nErrID 				=> udiErrID,
			iErrPos				=> usiErrPos,
		 );
		IF NOT xReadBusy THEN
			// allocate received module header
			stMDP_ModuleHeader	:= fbMDP_ReadModule.stMDP_ModuleHeader;
			// allocate information of startindexes in data buffer
			MEMCPY(ADR(arrStartIdx), ADR(fbMDP_ReadModule.arrStartIdx), SIZEOF(arrStartIdx) );
			// reset module content struct
			MEMSET( ADR(stMDP_ModuleContent), 0, SIZEOF(stMDP_ModuleContent) );
			// allocate received data to NIC struct
			stMDP_ModuleContent.uiLen		:= arrData[0];
			MEMCPY(ADR(stMDP_ModuleContent.sMainboard1p05v),			ADR(arrData)+arrStartIdx[1],	MIN(arrStartIdx[2]-arrStartIdx[1],	SIZEOF(stMDP_ModuleContent.sMainboard1p05v))     );
			MEMCPY(ADR(stMDP_ModuleContent.sMainboardVccCore),			ADR(arrData)+arrStartIdx[2],	MIN(arrStartIdx[3]-arrStartIdx[2],	SIZEOF(stMDP_ModuleContent.sMainboardVccCore))     );
			MEMCPY(ADR(stMDP_ModuleContent.sMainboard5v),				ADR(arrData)+arrStartIdx[3],	MIN(arrStartIdx[4]-arrStartIdx[3],	SIZEOF(stMDP_ModuleContent.sMainboard5v))     );
			MEMCPY(ADR(stMDP_ModuleContent.sMainboard12v),				ADR(arrData)+arrStartIdx[4],	MIN(arrStartIdx[5]-arrStartIdx[4],	SIZEOF(stMDP_ModuleContent.sMainboard12v))     );
			MEMCPY(ADR(stMDP_ModuleContent.sMainboardVBatt),			ADR(arrData)+arrStartIdx[5],	MIN(arrStartIdx[6]-arrStartIdx[5],	SIZEOF(stMDP_ModuleContent.sMainboardVBatt))     );
			MEMCPY(ADR(stMDP_ModuleContent.sMainboardPwrCtrlVcc),		ADR(arrData)+arrStartIdx[6],	MIN(arrStartIdx[7]-arrStartIdx[6],	SIZEOF(stMDP_ModuleContent.sMainboardPwrCtrlVcc))     );
			MEMCPY(ADR(stMDP_ModuleContent.sMainboardCX2100_5v),		ADR(arrData)+arrStartIdx[7],	MIN(arrStartIdx[8]-arrStartIdx[7],	SIZEOF(stMDP_ModuleContent.sMainboardCX2100_5v))     );
			MEMCPY(ADR(stMDP_ModuleContent.sMainboardCX2100_12v),		ADR(arrData)+arrStartIdx[8],	MIN(arrStartIdx[9]-arrStartIdx[8],	SIZEOF(stMDP_ModuleContent.sMainboardCX2100_12v))     );
			MEMCPY(ADR(stMDP_ModuleContent.sMainboardCX2100_24v),		ADR(arrData)+arrStartIdx[9],	MIN(arrStartIdx[10]-arrStartIdx[9],	SIZEOF(stMDP_ModuleContent.sMainboardCX2100_24v))     );

			// reset FB
			xBusy 				:= FALSE;
		END_IF
	END_IF

	// check timeout
	TimeOut();
	IF TimeOut.Q THEN
		TimeOut(IN 				:= FALSE);
		xError					:= TRUE;
		udiErrID				:= INT_TO_UINT(eMDP_Err_PLC) * 16#10000 + INT_TO_UINT(eMDP_ErrPLC_TimeOut);
	END_IF
END_IF

IF xError THEN
	// reset FB
	xBusy 						:= FALSE;
END_IF

END_FUNCTION_BLOCK

// ---- POUs/MDP_Function_Blocks/FB_MDP_Mainboard_ReadTBL4.TcPOU
FUNCTION_BLOCK FB_MDP_Mainboard_ReadTBL4

VAR_INPUT
	xExecute				: BOOL;								// Function block execution is triggered by a rising edge at this input
	tTimeout				: TIME		:= DEFAULT_ADS_TIMEOUT;	// States the time before the function is cancelled
	usiModIdx				: USINT		:= 0;					// Index number of chosen MDP device
	sAmsNetId				: T_AmsNetId;						// keep empty '' for the local device
END_VAR

VAR_OUTPUT
	xBusy					: BOOL;
	xError					: BOOL;
	udiErrID				: UDINT;
	usiErrPos				: USINT;							// If a subindex is not supported, iErrPos indicates at which subindex the error appears first
	stMDP_ModuleHeader		: ST_MDP_ModuleHeader;
	stMDP_ModuleContent		: ST_MDP_MainboardTBL4;	
END_VAR

VAR
	fbMDP_ReadModule		: FB_MDP_ReadModule;
	arrData					: ARRAY[0..70] OF BYTE;				// requested data
	arrStartIdx				: ARRAY[0..11] OF UINT;				// startindexes in bytes of each subindex element

	stMDP_Addr				: ST_MDP_Addr;
	eModuleType				: E_MDP_ModuleType;
	usiSubIdxCount			: USINT;

	xSubExecute				: BOOL;
	xReadBusy				: BOOL;

	RisingEdge				: R_TRIG;
	TimeOut					: TON;								// general timeout	
END_VAR

RisingEdge( CLK					:= xExecute );
IF NOT xBusy THEN											// FB only react to the external execute if it is not busy
	IF RisingEdge.Q THEN
		xBusy					:= TRUE;
		// reset variables
		xError					:= FALSE;
		udiErrID				:= 0;
		usiErrPos				:= 0;
		xSubExecute				:= TRUE;

		// specific values for Mainboard content
		stMDP_Addr.nArea		:= 16#08;
//		stMDP_Addr.nModuleId;								will be allocated dynamically
		stMDP_Addr.nTableId		:= 16#05; 					// Table4 is Location, Table5 is actual voltages, Table6 is nominal voltages - only need Table5
//		stMDP_Addr.nFlag;									not used up to now
//		stMDP_Addr.nSubIdx;									all subindexes will be requested
		eModuleType				:= eMDP_ModT_Mainboard;
		usiSubIdxCount			:= 10;						// TableId 16#01 contains 9 elements

		MEMSET( ADR(arrData), 0, SIZEOF(arrData) );			// reset buffer

		TimeOut(IN 				:= FALSE);
		TimeOut(PT 				:= tTimeout, IN 	:= TRUE);
	END_IF
END_IF


IF xBusy THEN
	IF xSubExecute THEN
		xSubExecute 			:= FALSE;

		fbMDP_ReadModule( bExecute := FALSE );
		fbMDP_ReadModule(
			stMDP_Addr			:= stMDP_Addr,
			eModuleType			:= eModuleType,
			iModIdx				:= usiModIdx,
			iSubIdxCount		:= usiSubIdxCount,
			bExecute			:= TRUE,
			tTimeout			:= tTimeout,
			pDstBuf				:= ADR(arrData),
			cbDstBufLen			:= SIZEOF(arrData),
			sAmsNetId			:= sAmsNetId,

			bBusy				=> xReadBusy,
			bError				=> xError,
			nErrID				=> udiErrID,
			iErrPos				=> usiErrPos,
			stMDP_DynAddr		=> ,
			iModuleTypeCount	=> ,
			iModuleCount		=> ,
			stMDP_ModuleHeader	=> ,
			arrStartIdx			=> ,
		);
	ELSE
		fbMDP_ReadModule(
			bExecute			:= FALSE,

			bBusy				=> xReadBusy,
			bError				=> xError,
			nErrID 				=> udiErrID,
			iErrPos				=> usiErrPos,
		 );
		IF NOT xReadBusy THEN
			// allocate received module header
			stMDP_ModuleHeader	:= fbMDP_ReadModule.stMDP_ModuleHeader;
			// allocate information of startindexes in data buffer
			MEMCPY(ADR(arrStartIdx), ADR(fbMDP_ReadModule.arrStartIdx), SIZEOF(arrStartIdx) );
			// reset module content struct
			MEMSET( ADR(stMDP_ModuleContent), 0, SIZEOF(stMDP_ModuleContent) );
			// allocate received data to NIC struct
			stMDP_ModuleContent.uiLen		:= arrData[0];
			MEMCPY(ADR(stMDP_ModuleContent.iMainboard1p05v),			ADR(arrData)+arrStartIdx[1],	MIN(arrStartIdx[2]-arrStartIdx[1],	SIZEOF(stMDP_ModuleContent.iMainboard1p05v))     );
			MEMCPY(ADR(stMDP_ModuleContent.iMainboardVccCore),			ADR(arrData)+arrStartIdx[2],	MIN(arrStartIdx[3]-arrStartIdx[2],	SIZEOF(stMDP_ModuleContent.iMainboardVccCore))     );
			MEMCPY(ADR(stMDP_ModuleContent.iMainboard5v),				ADR(arrData)+arrStartIdx[3],	MIN(arrStartIdx[4]-arrStartIdx[3],	SIZEOF(stMDP_ModuleContent.iMainboard5v))     );
			MEMCPY(ADR(stMDP_ModuleContent.iMainboard12v),				ADR(arrData)+arrStartIdx[4],	MIN(arrStartIdx[5]-arrStartIdx[4],	SIZEOF(stMDP_ModuleContent.iMainboard12v))     );
			MEMCPY(ADR(stMDP_ModuleContent.iMainboardVBatt),			ADR(arrData)+arrStartIdx[5],	MIN(arrStartIdx[6]-arrStartIdx[5],	SIZEOF(stMDP_ModuleContent.iMainboardVBatt))     );
			MEMCPY(ADR(stMDP_ModuleContent.iMainboardPwrCtrlVcc),		ADR(arrData)+arrStartIdx[6],	MIN(arrStartIdx[7]-arrStartIdx[6],	SIZEOF(stMDP_ModuleContent.iMainboardPwrCtrlVcc))     );
			MEMCPY(ADR(stMDP_ModuleContent.iMainboardCX2100_5v),		ADR(arrData)+arrStartIdx[7],	MIN(arrStartIdx[8]-arrStartIdx[7],	SIZEOF(stMDP_ModuleContent.iMainboardCX2100_5v))     );
			MEMCPY(ADR(stMDP_ModuleContent.iMainboardCX2100_12v),		ADR(arrData)+arrStartIdx[8],	MIN(arrStartIdx[9]-arrStartIdx[8],	SIZEOF(stMDP_ModuleContent.iMainboardCX2100_12v))     );
			MEMCPY(ADR(stMDP_ModuleContent.iMainboardCX2100_24v),		ADR(arrData)+arrStartIdx[9],	MIN(arrStartIdx[10]-arrStartIdx[9],	SIZEOF(stMDP_ModuleContent.iMainboardCX2100_24v))     );

			// reset FB
			xBusy 				:= FALSE;
		END_IF
	END_IF

	// check timeout
	TimeOut();
	IF TimeOut.Q THEN
		TimeOut(IN 				:= FALSE);
		xError					:= TRUE;
		udiErrID				:= INT_TO_UINT(eMDP_Err_PLC) * 16#10000 + INT_TO_UINT(eMDP_ErrPLC_TimeOut);
	END_IF
END_IF

IF xError THEN
	// reset FB
	xBusy 						:= FALSE;
END_IF

END_FUNCTION_BLOCK

// ---- POUs/MDP_Function_Blocks/FB_MDP_Time_ReadTBL1.TcPOU
FUNCTION_BLOCK FB_MDP_Time_ReadTBL1

VAR_INPUT
	xExecute				: BOOL;								// Function block execution is triggered by a rising edge at this input
	tTimeout				: TIME		:= DEFAULT_ADS_TIMEOUT;	// States the time before the function is cancelled
	usiModIdx				: USINT		:= 0;					// Index number of chosen MDP device
	sAmsNetId				: T_AmsNetId;						// keep empty '' for the local device
END_VAR

VAR_OUTPUT
	xBusy					: BOOL;
	xError					: BOOL;
	udiErrID				: UDINT;
	usiErrPos				: USINT;							// If a subindex is not supported, iErrPos indicates at which subindex the error appears first
	stMDP_ModuleHeader		: ST_MDP_ModuleHeader;
	stMDP_ModuleContent		: ST_MDP_TimeTBL1;	
END_VAR

VAR
	fbMDP_ReadModule		: FB_MDP_ReadModule;
	arrData					: ARRAY[0..42] OF BYTE;				// requested data
	arrStartIdx				: ARRAY[0..7] OF UINT;				// startindexes in bytes of each subindex element

	stMDP_Addr				: ST_MDP_Addr;
	eModuleType				: E_MDP_ModuleType;
	usiSubIdxCount			: USINT;

	xSubExecute				: BOOL;
	xReadBusy				: BOOL;

	RisingEdge				: R_TRIG;
	TimeOut					: TON;								// general timeout	
END_VAR

RisingEdge( CLK					:= xExecute );
IF NOT xBusy THEN										// FB only react to the external execute if it is not busy
	IF RisingEdge.Q THEN
		xBusy					:= TRUE;

		// reset variables
		xError					:= FALSE;
		udiErrID				:= 0;
		usiErrPos				:= 0;
		xSubExecute				:= TRUE;

		// specific values for Mainboard content
		stMDP_Addr.nArea		:= 16#08;
//		stMDP_Addr.nModuleId;							will be allocated dynamically
		stMDP_Addr.nTableId		:= 16#01;
//		stMDP_Addr.nFlag;								not used up to now
//		stMDP_Addr.nSubIdx;								all subindexes will be requested
		eModuleType				:= eMDP_ModT_Time;
		usiSubIdxCount			:= 6;					// TableId 16#01 contains 5 elements

		MEMSET( ADR(arrData), 0, SIZEOF(arrData) );		// reset buffer

		TimeOut(IN 				:= FALSE);
		TimeOut(PT 				:= tTimeout, IN 	:= TRUE);
	END_IF
END_IF


IF xBusy THEN
	IF xSubExecute THEN
		xSubExecute 			:= FALSE;

		fbMDP_ReadModule( bExecute := FALSE );
		fbMDP_ReadModule(
			stMDP_Addr			:= stMDP_Addr,
			eModuleType			:= eModuleType,
			iModIdx				:= usiModIdx,
			iSubIdxCount		:= usiSubIdxCount,
			bExecute			:= TRUE,
			tTimeout			:= tTimeout,
			pDstBuf				:= ADR(arrData),
			cbDstBufLen			:= SIZEOF(arrData),
			sAmsNetId			:= sAmsNetId,

			bBusy				=> xReadBusy,
			bError				=> xError,
			nErrID				=> udiErrID,
			iErrPos				=> usiErrPos,
			stMDP_DynAddr		=> ,
			iModuleTypeCount	=> ,
			iModuleCount		=> ,
			stMDP_ModuleHeader	=> ,
			arrStartIdx			=> ,
		);
	ELSE
		fbMDP_ReadModule(
			bExecute			:= FALSE,

			bBusy				=> xReadBusy,
			bError				=> xError,
			nErrID 				=> udiErrID,
			iErrPos				=> usiErrPos,
		 );
		IF NOT xReadBusy THEN
			// allocate received module header
			stMDP_ModuleHeader	:= fbMDP_ReadModule.stMDP_ModuleHeader;
			// allocate information of startindexes in data buffer
			MEMCPY(ADR(arrStartIdx), ADR(fbMDP_ReadModule.arrStartIdx), SIZEOF(arrStartIdx) );
			// reset module content struct
			MEMSET( ADR(stMDP_ModuleContent), 0, SIZEOF(stMDP_ModuleContent) );
			// allocate received data to NIC struct
			stMDP_ModuleContent.uiLen		:= arrData[0];
			MEMCPY(ADR(stMDP_ModuleContent.sSNTP_Server),				ADR(arrData)+arrStartIdx[1],	MIN(arrStartIdx[2]-arrStartIdx[1],	SIZEOF(stMDP_ModuleContent.sSNTP_Server))     );
			MEMCPY(ADR(stMDP_ModuleContent.udiSNTP_Refresh),			ADR(arrData)+arrStartIdx[2],	MIN(arrStartIdx[3]-arrStartIdx[2],	SIZEOF(stMDP_ModuleContent.udiSNTP_Refresh))     );
			MEMCPY(ADR(stMDP_ModuleContent.udiSec_Since_1_1_1970),		ADR(arrData)+arrStartIdx[3],	MIN(arrStartIdx[4]-arrStartIdx[3],	SIZEOF(stMDP_ModuleContent.udiSec_Since_1_1_1970))     );
			MEMCPY(ADR(stMDP_ModuleContent.sDateTime_Presentation),		ADR(arrData)+arrStartIdx[4],	MIN(arrStartIdx[5]-arrStartIdx[4],	SIZEOF(stMDP_ModuleContent.sDateTime_Presentation))     );
			MEMCPY(ADR(stMDP_ModuleContent.uiTimezone),					ADR(arrData)+arrStartIdx[5],	MIN(arrStartIdx[6]-arrStartIdx[5],	SIZEOF(stMDP_ModuleContent.uiTimezone))     );

			// reset FB
			xBusy 				:= FALSE;
		END_IF
	END_IF

	// check timeout
	TimeOut();
	IF TimeOut.Q THEN
		TimeOut(IN 				:= FALSE);
		xError					:= TRUE;
		udiErrID				:= INT_TO_UINT(eMDP_Err_PLC) * 16#10000 + INT_TO_UINT(eMDP_ErrPLC_TimeOut);
	END_IF
END_IF

IF xError THEN
	// reset FB
	xBusy 						:= FALSE;
END_IF

END_FUNCTION_BLOCK

// ---- POUs/MDP_Function_Blocks/FB_MDP_Time_ReadTBL2.TcPOU
FUNCTION_BLOCK FB_MDP_Time_ReadTBL2

VAR_INPUT
	xExecute				: BOOL;								// Function block execution is triggered by a rising edge at this input
	tTimeout				: TIME		:= DEFAULT_ADS_TIMEOUT;	// States the time before the function is cancelled
	usiModIdx				: USINT		:= 0;					// Index number of chosen MDP device
	sAmsNetId				: T_AmsNetId;						// keep empty '' for the local device
END_VAR

VAR_OUTPUT
	xBusy					: BOOL;
	xError					: BOOL;
	udiErrID				: UDINT;
	usiErrPos				: USINT;							// If a subindex is not supported, iErrPos indicates at which subindex the error appears first
	stMDP_ModuleHeader		: ST_MDP_ModuleHeader;
	stMDP_ModuleContent		: ST_MDP_TimeTBL2;	
END_VAR

VAR
	fbMDP_ReadModule		: FB_MDP_ReadModule;
	arrData					: ARRAY[0..3000] OF BYTE;				// requested data
	arrStartIdx				: ARRAY[0..102] OF UINT;				// startindexes in bytes of each subindex element

	stMDP_Addr				: ST_MDP_Addr;
	eModuleType				: E_MDP_ModuleType;
	usiSubIdxCount			: USINT;

	xSubExecute				: BOOL;
	xReadBusy				: BOOL;

	RisingEdge				: R_TRIG;
	TimeOut					: TON;								// general timeout	
END_VAR

RisingEdge( CLK					:= xExecute );
IF NOT xBusy THEN										// FB only react to the external execute if it is not busy
	IF RisingEdge.Q THEN
		xBusy					:= TRUE;

		// reset variables
		xError					:= FALSE;
		udiErrID				:= 0;
		usiErrPos				:= 0;
		xSubExecute				:= TRUE;

		// specific values for Mainboard content
		stMDP_Addr.nArea		:= 16#08;
//		stMDP_Addr.nModuleId;							will be allocated dynamically
		stMDP_Addr.nTableId		:= 16#02;
//		stMDP_Addr.nFlag;								not used up to now
//		stMDP_Addr.nSubIdx;								all subindexes will be requested
		eModuleType				:= eMDP_ModT_Time;
		usiSubIdxCount			:= 102;					// TableId 16#01 contains 101 elements

		MEMSET( ADR(arrData), 0, SIZEOF(arrData) );		// reset buffer

		TimeOut(IN 				:= FALSE);
		TimeOut(PT 				:= tTimeout, IN 	:= TRUE);
	END_IF
END_IF


IF xBusy THEN
	IF xSubExecute THEN
		xSubExecute 			:= FALSE;

		fbMDP_ReadModule( bExecute := FALSE );
		fbMDP_ReadModule(
			stMDP_Addr			:= stMDP_Addr,
			eModuleType			:= eModuleType,
			iModIdx				:= usiModIdx,
			iSubIdxCount		:= usiSubIdxCount,
			bExecute			:= TRUE,
			tTimeout			:= tTimeout,
			pDstBuf				:= ADR(arrData),
			cbDstBufLen			:= SIZEOF(arrData),
			sAmsNetId			:= sAmsNetId,

			bBusy				=> xReadBusy,
			bError				=> xError,
			nErrID				=> udiErrID,
			iErrPos				=> usiErrPos,
			stMDP_DynAddr		=> ,
			iModuleTypeCount	=> ,
			iModuleCount		=> ,
			stMDP_ModuleHeader	=> ,
			arrStartIdx			=> ,
		);
	ELSE
		fbMDP_ReadModule(
			bExecute			:= FALSE,

			bBusy				=> xReadBusy,
			bError				=> xError,
			nErrID 				=> udiErrID,
			iErrPos				=> usiErrPos,
		 );
		IF NOT xReadBusy THEN
			// allocate received module header
			stMDP_ModuleHeader	:= fbMDP_ReadModule.stMDP_ModuleHeader;
			// allocate information of startindexes in data buffer
			MEMCPY(ADR(arrStartIdx), ADR(fbMDP_ReadModule.arrStartIdx), SIZEOF(arrStartIdx) );
			// reset module content struct
			MEMSET( ADR(stMDP_ModuleContent), 0, SIZEOF(stMDP_ModuleContent) );
			// allocate received data to NIC struct
			stMDP_ModuleContent.uiLen		:= arrData[0];
			MEMCPY(ADR(stMDP_ModuleContent.sTimezone1),		ADR(arrData)+arrStartIdx[1],	MIN(arrStartIdx[2]-arrStartIdx[1],		SIZEOF(stMDP_ModuleContent.sTimezone1))     );
			MEMCPY(ADR(stMDP_ModuleContent.sTimezone2),		ADR(arrData)+arrStartIdx[2],	MIN(arrStartIdx[3]-arrStartIdx[2],		SIZEOF(stMDP_ModuleContent.sTimezone2))     );
			MEMCPY(ADR(stMDP_ModuleContent.sTimezone3),		ADR(arrData)+arrStartIdx[3],	MIN(arrStartIdx[4]-arrStartIdx[3],		SIZEOF(stMDP_ModuleContent.sTimezone3))     );
			MEMCPY(ADR(stMDP_ModuleContent.sTimezone4),		ADR(arrData)+arrStartIdx[4],	MIN(arrStartIdx[5]-arrStartIdx[4],		SIZEOF(stMDP_ModuleContent.sTimezone4))     );
			MEMCPY(ADR(stMDP_ModuleContent.sTimezone5),		ADR(arrData)+arrStartIdx[5],	MIN(arrStartIdx[6]-arrStartIdx[5],		SIZEOF(stMDP_ModuleContent.sTimezone5))     );
			MEMCPY(ADR(stMDP_ModuleContent.sTimezone6),		ADR(arrData)+arrStartIdx[6],	MIN(arrStartIdx[7]-arrStartIdx[6],		SIZEOF(stMDP_ModuleContent.sTimezone6))     );
			MEMCPY(ADR(stMDP_ModuleContent.sTimezone7),		ADR(arrData)+arrStartIdx[7],	MIN(arrStartIdx[8]-arrStartIdx[7],		SIZEOF(stMDP_ModuleContent.sTimezone7))     );
			MEMCPY(ADR(stMDP_ModuleContent.sTimezone8),		ADR(arrData)+arrStartIdx[8],	MIN(arrStartIdx[9]-arrStartIdx[8],		SIZEOF(stMDP_ModuleContent.sTimezone8))     );
			MEMCPY(ADR(stMDP_ModuleContent.sTimezone9),		ADR(arrData)+arrStartIdx[9],	MIN(arrStartIdx[10]-arrStartIdx[9],		SIZEOF(stMDP_ModuleContent.sTimezone9))     );
			MEMCPY(ADR(stMDP_ModuleContent.sTimezone10),	ADR(arrData)+arrStartIdx[10],	MIN(arrStartIdx[11]-arrStartIdx[10],	SIZEOF(stMDP_ModuleContent.sTimezone10))     );
			MEMCPY(ADR(stMDP_ModuleContent.sTimezone11),	ADR(arrData)+arrStartIdx[11],	MIN(arrStartIdx[12]-arrStartIdx[11],	SIZEOF(stMDP_ModuleContent.sTimezone11))     );
			MEMCPY(ADR(stMDP_ModuleContent.sTimezone12),	ADR(arrData)+arrStartIdx[12],	MIN(arrStartIdx[13]-arrStartIdx[12],	SIZEOF(stMDP_ModuleContent.sTimezone12))     );
			MEMCPY(ADR(stMDP_ModuleContent.sTimezone13),	ADR(arrData)+arrStartIdx[13],	MIN(arrStartIdx[14]-arrStartIdx[13],	SIZEOF(stMDP_ModuleContent.sTimezone13))     );
			MEMCPY(ADR(stMDP_ModuleContent.sTimezone14),	ADR(arrData)+arrStartIdx[14],	MIN(arrStartIdx[15]-arrStartIdx[14],	SIZEOF(stMDP_ModuleContent.sTimezone14))     );
			MEMCPY(ADR(stMDP_ModuleContent.sTimezone15),	ADR(arrData)+arrStartIdx[15],	MIN(arrStartIdx[16]-arrStartIdx[15],	SIZEOF(stMDP_ModuleContent.sTimezone15))     );
			MEMCPY(ADR(stMDP_ModuleContent.sTimezone16),	ADR(arrData)+arrStartIdx[16],	MIN(arrStartIdx[17]-arrStartIdx[16],	SIZEOF(stMDP_ModuleContent.sTimezone16))     );
			MEMCPY(ADR(stMDP_ModuleContent.sTimezone17),	ADR(arrData)+arrStartIdx[17],	MIN(arrStartIdx[18]-arrStartIdx[17],	SIZEOF(stMDP_ModuleContent.sTimezone17))     );
			MEMCPY(ADR(stMDP_ModuleContent.sTimezone18),	ADR(arrData)+arrStartIdx[18],	MIN(arrStartIdx[19]-arrStartIdx[18],	SIZEOF(stMDP_ModuleContent.sTimezone18))     );
			MEMCPY(ADR(stMDP_ModuleContent.sTimezone19),	ADR(arrData)+arrStartIdx[19],	MIN(arrStartIdx[20]-arrStartIdx[19],	SIZEOF(stMDP_ModuleContent.sTimezone19))     );
			MEMCPY(ADR(stMDP_ModuleContent.sTimezone20),	ADR(arrData)+arrStartIdx[20],	MIN(arrStartIdx[21]-arrStartIdx[20],	SIZEOF(stMDP_ModuleContent.sTimezone20))     );
			MEMCPY(ADR(stMDP_ModuleContent.sTimezone21),	ADR(arrData)+arrStartIdx[21],	MIN(arrStartIdx[22]-arrStartIdx[21],	SIZEOF(stMDP_ModuleContent.sTimezone21))     );
			MEMCPY(ADR(stMDP_ModuleContent.sTimezone22),	ADR(arrData)+arrStartIdx[22],	MIN(arrStartIdx[23]-arrStartIdx[22],	SIZEOF(stMDP_ModuleContent.sTimezone22))     );
			MEMCPY(ADR(stMDP_ModuleContent.sTimezone23),	ADR(arrData)+arrStartIdx[23],	MIN(arrStartIdx[24]-arrStartIdx[23],	SIZEOF(stMDP_ModuleContent.sTimezone23))     );
			MEMCPY(ADR(stMDP_ModuleContent.sTimezone24),	ADR(arrData)+arrStartIdx[24],	MIN(arrStartIdx[25]-arrStartIdx[24],	SIZEOF(stMDP_ModuleContent.sTimezone24))     );
			MEMCPY(ADR(stMDP_ModuleContent.sTimezone25),	ADR(arrData)+arrStartIdx[25],	MIN(arrStartIdx[26]-arrStartIdx[25],	SIZEOF(stMDP_ModuleContent.sTimezone25))     );
			MEMCPY(ADR(stMDP_ModuleContent.sTimezone26),	ADR(arrData)+arrStartIdx[26],	MIN(arrStartIdx[27]-arrStartIdx[26],	SIZEOF(stMDP_ModuleContent.sTimezone26))     );
			MEMCPY(ADR(stMDP_ModuleContent.sTimezone27),	ADR(arrData)+arrStartIdx[27],	MIN(arrStartIdx[28]-arrStartIdx[27],	SIZEOF(stMDP_ModuleContent.sTimezone27))     );
			MEMCPY(ADR(stMDP_ModuleContent.sTimezone28),	ADR(arrData)+arrStartIdx[28],	MIN(arrStartIdx[29]-arrStartIdx[28],	SIZEOF(stMDP_ModuleContent.sTimezone28))     );
			MEMCPY(ADR(stMDP_ModuleContent.sTimezone29),	ADR(arrData)+arrStartIdx[29],	MIN(arrStartIdx[30]-arrStartIdx[29],	SIZEOF(stMDP_ModuleContent.sTimezone29))     );
			MEMCPY(ADR(stMDP_ModuleContent.sTimezone30),	ADR(arrData)+arrStartIdx[30],	MIN(arrStartIdx[31]-arrStartIdx[30],	SIZEOF(stMDP_ModuleContent.sTimezone30))     );			
			MEMCPY(ADR(stMDP_ModuleContent.sTimezone31),	ADR(arrData)+arrStartIdx[31],	MIN(arrStartIdx[32]-arrStartIdx[31],	SIZEOF(stMDP_ModuleContent.sTimezone31))     );
			MEMCPY(ADR(stMDP_ModuleContent.sTimezone32),	ADR(arrData)+arrStartIdx[32],	MIN(arrStartIdx[33]-arrStartIdx[32],	SIZEOF(stMDP_ModuleContent.sTimezone32))     );
			MEMCPY(ADR(stMDP_ModuleContent.sTimezone33),	ADR(arrData)+arrStartIdx[33],	MIN(arrStartIdx[34]-arrStartIdx[33],	SIZEOF(stMDP_ModuleContent.sTimezone33))     );
			MEMCPY(ADR(stMDP_ModuleContent.sTimezone34),	ADR(arrData)+arrStartIdx[34],	MIN(arrStartIdx[35]-arrStartIdx[34],	SIZEOF(stMDP_ModuleContent.sTimezone34))     );
			MEMCPY(ADR(stMDP_ModuleContent.sTimezone35),	ADR(arrData)+arrStartIdx[35],	MIN(arrStartIdx[36]-arrStartIdx[35],	SIZEOF(stMDP_ModuleContent.sTimezone35))     );
			MEMCPY(ADR(stMDP_ModuleContent.sTimezone36),	ADR(arrData)+arrStartIdx[36],	MIN(arrStartIdx[37]-arrStartIdx[36],	SIZEOF(stMDP_ModuleContent.sTimezone36))     );
			MEMCPY(ADR(stMDP_ModuleContent.sTimezone37),	ADR(arrData)+arrStartIdx[37],	MIN(arrStartIdx[38]-arrStartIdx[37],	SIZEOF(stMDP_ModuleContent.sTimezone37))     );
			MEMCPY(ADR(stMDP_ModuleContent.sTimezone38),	ADR(arrData)+arrStartIdx[38],	MIN(arrStartIdx[39]-arrStartIdx[38],	SIZEOF(stMDP_ModuleContent.sTimezone38))     );
			MEMCPY(ADR(stMDP_ModuleContent.sTimezone39),	ADR(arrData)+arrStartIdx[39],	MIN(arrStartIdx[40]-arrStartIdx[39],	SIZEOF(stMDP_ModuleContent.sTimezone39))     );
			MEMCPY(ADR(stMDP_ModuleContent.sTimezone40),	ADR(arrData)+arrStartIdx[40],	MIN(arrStartIdx[41]-arrStartIdx[40],	SIZEOF(stMDP_ModuleContent.sTimezone40))     );
			MEMCPY(ADR(stMDP_ModuleContent.sTimezone41),	ADR(arrData)+arrStartIdx[41],	MIN(arrStartIdx[42]-arrStartIdx[41],	SIZEOF(stMDP_ModuleContent.sTimezone41))     );
			MEMCPY(ADR(stMDP_ModuleContent.sTimezone42),	ADR(arrData)+arrStartIdx[42],	MIN(arrStartIdx[43]-arrStartIdx[42],	SIZEOF(stMDP_ModuleContent.sTimezone42))     );
			MEMCPY(ADR(stMDP_ModuleContent.sTimezone43),	ADR(arrData)+arrStartIdx[43],	MIN(arrStartIdx[44]-arrStartIdx[43],	SIZEOF(stMDP_ModuleContent.sTimezone43))     );
			MEMCPY(ADR(stMDP_ModuleContent.sTimezone44),	ADR(arrData)+arrStartIdx[44],	MIN(arrStartIdx[45]-arrStartIdx[44],	SIZEOF(stMDP_ModuleContent.sTimezone44))     );
			MEMCPY(ADR(stMDP_ModuleContent.sTimezone45),	ADR(arrData)+arrStartIdx[45],	MIN(arrStartIdx[46]-arrStartIdx[45],	SIZEOF(stMDP_ModuleContent.sTimezone45))     );
			MEMCPY(ADR(stMDP_ModuleContent.sTimezone46),	ADR(arrData)+arrStartIdx[46],	MIN(arrStartIdx[47]-arrStartIdx[46],	SIZEOF(stMDP_ModuleContent.sTimezone46))     );
			MEMCPY(ADR(stMDP_ModuleContent.sTimezone47),	ADR(arrData)+arrStartIdx[47],	MIN(arrStartIdx[48]-arrStartIdx[47],	SIZEOF(stMDP_ModuleContent.sTimezone47))     );
			MEMCPY(ADR(stMDP_ModuleContent.sTimezone48),	ADR(arrData)+arrStartIdx[48],	MIN(arrStartIdx[49]-arrStartIdx[48],	SIZEOF(stMDP_ModuleContent.sTimezone48))     );
			MEMCPY(ADR(stMDP_ModuleContent.sTimezone49),	ADR(arrData)+arrStartIdx[49],	MIN(arrStartIdx[50]-arrStartIdx[49],	SIZEOF(stMDP_ModuleContent.sTimezone49))     );
			MEMCPY(ADR(stMDP_ModuleContent.sTimezone50),	ADR(arrData)+arrStartIdx[50],	MIN(arrStartIdx[51]-arrStartIdx[50],	SIZEOF(stMDP_ModuleContent.sTimezone50))     );		
			MEMCPY(ADR(stMDP_ModuleContent.sTimezone51),	ADR(arrData)+arrStartIdx[51],	MIN(arrStartIdx[52]-arrStartIdx[51],	SIZEOF(stMDP_ModuleContent.sTimezone51))     );
			MEMCPY(ADR(stMDP_ModuleContent.sTimezone52),	ADR(arrData)+arrStartIdx[52],	MIN(arrStartIdx[53]-arrStartIdx[52],	SIZEOF(stMDP_ModuleContent.sTimezone52))     );
			MEMCPY(ADR(stMDP_ModuleContent.sTimezone53),	ADR(arrData)+arrStartIdx[53],	MIN(arrStartIdx[54]-arrStartIdx[53],	SIZEOF(stMDP_ModuleContent.sTimezone53))     );
			MEMCPY(ADR(stMDP_ModuleContent.sTimezone54),	ADR(arrData)+arrStartIdx[54],	MIN(arrStartIdx[55]-arrStartIdx[54],	SIZEOF(stMDP_ModuleContent.sTimezone54))     );
			MEMCPY(ADR(stMDP_ModuleContent.sTimezone55),	ADR(arrData)+arrStartIdx[55],	MIN(arrStartIdx[56]-arrStartIdx[55],	SIZEOF(stMDP_ModuleContent.sTimezone55))     );
			MEMCPY(ADR(stMDP_ModuleContent.sTimezone56),	ADR(arrData)+arrStartIdx[56],	MIN(arrStartIdx[57]-arrStartIdx[56],	SIZEOF(stMDP_ModuleContent.sTimezone56))     );
			MEMCPY(ADR(stMDP_ModuleContent.sTimezone57),	ADR(arrData)+arrStartIdx[57],	MIN(arrStartIdx[58]-arrStartIdx[57],	SIZEOF(stMDP_ModuleContent.sTimezone57))     );
			MEMCPY(ADR(stMDP_ModuleContent.sTimezone58),	ADR(arrData)+arrStartIdx[58],	MIN(arrStartIdx[59]-arrStartIdx[58],	SIZEOF(stMDP_ModuleContent.sTimezone58))     );
			MEMCPY(ADR(stMDP_ModuleContent.sTimezone59),	ADR(arrData)+arrStartIdx[59],	MIN(arrStartIdx[60]-arrStartIdx[59],	SIZEOF(stMDP_ModuleContent.sTimezone59))     );
			MEMCPY(ADR(stMDP_ModuleContent.sTimezone60),	ADR(arrData)+arrStartIdx[60],	MIN(arrStartIdx[61]-arrStartIdx[60],	SIZEOF(stMDP_ModuleContent.sTimezone60))     );
			MEMCPY(ADR(stMDP_ModuleContent.sTimezone61),	ADR(arrData)+arrStartIdx[61],	MIN(arrStartIdx[62]-arrStartIdx[61],	SIZEOF(stMDP_ModuleContent.sTimezone61))     );
			MEMCPY(ADR(stMDP_ModuleContent.sTimezone62),	ADR(arrData)+arrStartIdx[62],	MIN(arrStartIdx[63]-arrStartIdx[62],	SIZEOF(stMDP_ModuleContent.sTimezone62))     );
			MEMCPY(ADR(stMDP_ModuleContent.sTimezone63),	ADR(arrData)+arrStartIdx[63],	MIN(arrStartIdx[64]-arrStartIdx[63],	SIZEOF(stMDP_ModuleContent.sTimezone63))     );
			MEMCPY(ADR(stMDP_ModuleContent.sTimezone64),	ADR(arrData)+arrStartIdx[64],	MIN(arrStartIdx[65]-arrStartIdx[64],	SIZEOF(stMDP_ModuleContent.sTimezone64))     );
			MEMCPY(ADR(stMDP_ModuleContent.sTimezone65),	ADR(arrData)+arrStartIdx[65],	MIN(arrStartIdx[66]-arrStartIdx[65],	SIZEOF(stMDP_ModuleContent.sTimezone65))     );
			MEMCPY(ADR(stMDP_ModuleContent.sTimezone66),	ADR(arrData)+arrStartIdx[66],	MIN(arrStartIdx[67]-arrStartIdx[66],	SIZEOF(stMDP_ModuleContent.sTimezone66))     );
			MEMCPY(ADR(stMDP_ModuleContent.sTimezone67),	ADR(arrData)+arrStartIdx[67],	MIN(arrStartIdx[68]-arrStartIdx[67],	SIZEOF(stMDP_ModuleContent.sTimezone67))     );
			MEMCPY(ADR(stMDP_ModuleContent.sTimezone68),	ADR(arrData)+arrStartIdx[68],	MIN(arrStartIdx[69]-arrStartIdx[68],	SIZEOF(stMDP_ModuleContent.sTimezone68))     );
			MEMCPY(ADR(stMDP_ModuleContent.sTimezone69),	ADR(arrData)+arrStartIdx[69],	MIN(arrStartIdx[70]-arrStartIdx[69],	SIZEOF(stMDP_ModuleContent.sTimezone69))     );
			MEMCPY(ADR(stMDP_ModuleContent.sTimezone70),	ADR(arrData)+arrStartIdx[70],	MIN(arrStartIdx[71]-arrStartIdx[70],	SIZEOF(stMDP_ModuleContent.sTimezone70))     );			
			MEMCPY(ADR(stMDP_ModuleContent.sTimezone71),	ADR(arrData)+arrStartIdx[71],	MIN(arrStartIdx[72]-arrStartIdx[71],	SIZEOF(stMDP_ModuleContent.sTimezone71))     );
			MEMCPY(ADR(stMDP_ModuleContent.sTimezone72),	ADR(arrData)+arrStartIdx[72],	MIN(arrStartIdx[73]-arrStartIdx[72],	SIZEOF(stMDP_ModuleContent.sTimezone72))     );
			MEMCPY(ADR(stMDP_ModuleContent.sTimezone73),	ADR(arrData)+arrStartIdx[73],	MIN(arrStartIdx[74]-arrStartIdx[73],	SIZEOF(stMDP_ModuleContent.sTimezone73))     );
			MEMCPY(ADR(stMDP_ModuleContent.sTimezone74),	ADR(arrData)+arrStartIdx[74],	MIN(arrStartIdx[75]-arrStartIdx[74],	SIZEOF(stMDP_ModuleContent.sTimezone74))     );
			MEMCPY(ADR(stMDP_ModuleContent.sTimezone75),	ADR(arrData)+arrStartIdx[75],	MIN(arrStartIdx[76]-arrStartIdx[75],	SIZEOF(stMDP_ModuleContent.sTimezone75))     );
			MEMCPY(ADR(stMDP_ModuleContent.sTimezone76),	ADR(arrData)+arrStartIdx[76],	MIN(arrStartIdx[77]-arrStartIdx[76],	SIZEOF(stMDP_ModuleContent.sTimezone76))     );
			MEMCPY(ADR(stMDP_ModuleContent.sTimezone77),	ADR(arrData)+arrStartIdx[77],	MIN(arrStartIdx[78]-arrStartIdx[77],	SIZEOF(stMDP_ModuleContent.sTimezone77))     );
			MEMCPY(ADR(stMDP_ModuleContent.sTimezone78),	ADR(arrData)+arrStartIdx[78],	MIN(arrStartIdx[79]-arrStartIdx[78],	SIZEOF(stMDP_ModuleContent.sTimezone78))     );
			MEMCPY(ADR(stMDP_ModuleContent.sTimezone79),	ADR(arrData)+arrStartIdx[79],	MIN(arrStartIdx[80]-arrStartIdx[79],	SIZEOF(stMDP_ModuleContent.sTimezone79))     );
			MEMCPY(ADR(stMDP_ModuleContent.sTimezone80),	ADR(arrData)+arrStartIdx[80],	MIN(arrStartIdx[81]-arrStartIdx[80],	SIZEOF(stMDP_ModuleContent.sTimezone80))     );
			MEMCPY(ADR(stMDP_ModuleContent.sTimezone81),	ADR(arrData)+arrStartIdx[81],	MIN(arrStartIdx[82]-arrStartIdx[81],	SIZEOF(stMDP_ModuleContent.sTimezone81))     );
			MEMCPY(ADR(stMDP_ModuleContent.sTimezone82),	ADR(arrData)+arrStartIdx[82],	MIN(arrStartIdx[83]-arrStartIdx[82],	SIZEOF(stMDP_ModuleContent.sTimezone82))     );
			MEMCPY(ADR(stMDP_ModuleContent.sTimezone83),	ADR(arrData)+arrStartIdx[83],	MIN(arrStartIdx[84]-arrStartIdx[83],	SIZEOF(stMDP_ModuleContent.sTimezone83))     );
			MEMCPY(ADR(stMDP_ModuleContent.sTimezone84),	ADR(arrData)+arrStartIdx[84],	MIN(arrStartIdx[85]-arrStartIdx[84],	SIZEOF(stMDP_ModuleContent.sTimezone84))     );
			MEMCPY(ADR(stMDP_ModuleContent.sTimezone85),	ADR(arrData)+arrStartIdx[85],	MIN(arrStartIdx[86]-arrStartIdx[85],	SIZEOF(stMDP_ModuleContent.sTimezone85))     );
			MEMCPY(ADR(stMDP_ModuleContent.sTimezone86),	ADR(arrData)+arrStartIdx[86],	MIN(arrStartIdx[87]-arrStartIdx[86],	SIZEOF(stMDP_ModuleContent.sTimezone86))     );
			MEMCPY(ADR(stMDP_ModuleContent.sTimezone87),	ADR(arrData)+arrStartIdx[87],	MIN(arrStartIdx[88]-arrStartIdx[87],	SIZEOF(stMDP_ModuleContent.sTimezone87))     );
			MEMCPY(ADR(stMDP_ModuleContent.sTimezone88),	ADR(arrData)+arrStartIdx[88],	MIN(arrStartIdx[89]-arrStartIdx[88],	SIZEOF(stMDP_ModuleContent.sTimezone88))     );
			MEMCPY(ADR(stMDP_ModuleContent.sTimezone89),	ADR(arrData)+arrStartIdx[89],	MIN(arrStartIdx[90]-arrStartIdx[89],	SIZEOF(stMDP_ModuleContent.sTimezone89))     );
			MEMCPY(ADR(stMDP_ModuleContent.sTimezone90),	ADR(arrData)+arrStartIdx[90],	MIN(arrStartIdx[91]-arrStartIdx[90],	SIZEOF(stMDP_ModuleContent.sTimezone90))     );
			MEMCPY(ADR(stMDP_ModuleContent.sTimezone91),	ADR(arrData)+arrStartIdx[91],	MIN(arrStartIdx[92]-arrStartIdx[91],	SIZEOF(stMDP_ModuleContent.sTimezone91))     );
			MEMCPY(ADR(stMDP_ModuleContent.sTimezone92),	ADR(arrData)+arrStartIdx[92],	MIN(arrStartIdx[93]-arrStartIdx[92],	SIZEOF(stMDP_ModuleContent.sTimezone92))     );
			MEMCPY(ADR(stMDP_ModuleContent.sTimezone93),	ADR(arrData)+arrStartIdx[93],	MIN(arrStartIdx[94]-arrStartIdx[93],	SIZEOF(stMDP_ModuleContent.sTimezone93))     );
			MEMCPY(ADR(stMDP_ModuleContent.sTimezone94),	ADR(arrData)+arrStartIdx[94],	MIN(arrStartIdx[95]-arrStartIdx[94],	SIZEOF(stMDP_ModuleContent.sTimezone94))     );
			MEMCPY(ADR(stMDP_ModuleContent.sTimezone95),	ADR(arrData)+arrStartIdx[95],	MIN(arrStartIdx[96]-arrStartIdx[95],	SIZEOF(stMDP_ModuleContent.sTimezone95))     );
			MEMCPY(ADR(stMDP_ModuleContent.sTimezone96),	ADR(arrData)+arrStartIdx[96],	MIN(arrStartIdx[97]-arrStartIdx[96],	SIZEOF(stMDP_ModuleContent.sTimezone96))     );
			MEMCPY(ADR(stMDP_ModuleContent.sTimezone97),	ADR(arrData)+arrStartIdx[97],	MIN(arrStartIdx[98]-arrStartIdx[97],	SIZEOF(stMDP_ModuleContent.sTimezone97))     );
			MEMCPY(ADR(stMDP_ModuleContent.sTimezone98),	ADR(arrData)+arrStartIdx[98],	MIN(arrStartIdx[99]-arrStartIdx[98],	SIZEOF(stMDP_ModuleContent.sTimezone98))     );
			MEMCPY(ADR(stMDP_ModuleContent.sTimezone99),	ADR(arrData)+arrStartIdx[99],	MIN(arrStartIdx[100]-arrStartIdx[99],	SIZEOF(stMDP_ModuleContent.sTimezone99))     );
			MEMCPY(ADR(stMDP_ModuleContent.sTimezone100),	ADR(arrData)+arrStartIdx[100],	MIN(arrStartIdx[101]-arrStartIdx[100],	SIZEOF(stMDP_ModuleContent.sTimezone100))     );
			MEMCPY(ADR(stMDP_ModuleContent.sTimezone101),	ADR(arrData)+arrStartIdx[101],	MIN(arrStartIdx[102]-arrStartIdx[101],	SIZEOF(stMDP_ModuleContent.sTimezone101))     );

			// reset FB
			xBusy 				:= FALSE;
		END_IF
	END_IF

	// check timeout
	TimeOut();
	IF TimeOut.Q THEN
		TimeOut(IN 				:= FALSE);
		xError					:= TRUE;
		udiErrID				:= INT_TO_UINT(eMDP_Err_PLC) * 16#10000 + INT_TO_UINT(eMDP_ErrPLC_TimeOut);
	END_IF
END_IF

IF xError THEN
	// reset FB
	xBusy 						:= FALSE;
END_IF

END_FUNCTION_BLOCK

// ---- POUs/MDP_Function_Blocks/FB_MDP_Memory_ReadTBL1.TcPOU
FUNCTION_BLOCK FB_MDP_Memory_ReadTBL1

VAR_INPUT
	xExecute				: BOOL;								// Function block execution is triggered by a rising edge at this input
	tTimeout				: TIME		:= DEFAULT_ADS_TIMEOUT;	// States the time before the function is cancelled
	usiModIdx				: USINT		:= 0;					// Index number of chosen MDP device
	sAmsNetId				: T_AmsNetId;						// keep empty '' for the local device
END_VAR

VAR_OUTPUT
	xBusy					: BOOL;
	xError					: BOOL;
	udiErrID				: UDINT;
	usiErrPos				: USINT;							// If a subindex is not supported, iErrPos indicates at which subindex the error appears first
	stMDP_ModuleHeader		: ST_MDP_ModuleHeader;
	stMDP_ModuleContent		: ST_MDP_MemoryTBL1;	
END_VAR

VAR
	fbMDP_ReadModule		: FB_MDP_ReadModule;
	arrData					: ARRAY[0..10] OF BYTE;			// requested data
	arrStartIdx				: ARRAY[0..7] OF UINT;				// startindexes in bytes of each subindex element

	stMDP_Addr				: ST_MDP_Addr;
	eModuleType				: E_MDP_ModuleType;
	usiSubIdxCount			: USINT;

	xSubExecute				: BOOL;
	xReadBusy				: BOOL;

	RisingEdge				: R_TRIG;
	TimeOut					: TON;								// general timeout	
END_VAR

RisingEdge( CLK					:= xExecute );
IF NOT xBusy THEN										// FB only react to the external execute if it is not busy
	IF RisingEdge.Q THEN
		xBusy					:= TRUE;

		// reset variables
		xError					:= FALSE;
		udiErrID				:= 0;
		usiErrPos				:= 0;
		xSubExecute				:= TRUE;

		// specific values for Mainboard content
		stMDP_Addr.nArea		:= 16#08;
//		stMDP_Addr.nModuleId;							will be allocated dynamically
		stMDP_Addr.nTableId		:= 16#01;
//		stMDP_Addr.nFlag;								not used up to now
//		stMDP_Addr.nSubIdx;								all subindexes will be requested
		eModuleType				:= eMDP_ModT_Memory;
		usiSubIdxCount			:= 6;					// TableId 16#01 contains 5 elements

		MEMSET( ADR(arrData), 0, SIZEOF(arrData) );		// reset buffer

		TimeOut(IN 				:= FALSE);
		TimeOut(PT 				:= tTimeout, IN 	:= TRUE);
	END_IF
END_IF


IF xBusy THEN
	IF xSubExecute THEN
		xSubExecute 			:= FALSE;

		fbMDP_ReadModule( bExecute := FALSE );
		fbMDP_ReadModule(
			stMDP_Addr			:= stMDP_Addr,
			eModuleType			:= eModuleType,
			iModIdx				:= usiModIdx,
			iSubIdxCount		:= usiSubIdxCount,
			bExecute			:= TRUE,
			tTimeout			:= tTimeout,
			pDstBuf				:= ADR(arrData),
			cbDstBufLen			:= SIZEOF(arrData),
			sAmsNetId			:= sAmsNetId,

			bBusy				=> xReadBusy,
			bError				=> xError,
			nErrID				=> udiErrID,
			iErrPos				=> usiErrPos,
			stMDP_DynAddr		=> ,
			iModuleTypeCount	=> ,
			iModuleCount		=> ,
			stMDP_ModuleHeader	=> ,
			arrStartIdx			=> ,
		);
	ELSE
		fbMDP_ReadModule(
			bExecute			:= FALSE,

			bBusy				=> xReadBusy,
			bError				=> xError,
			nErrID 				=> udiErrID,
			iErrPos				=> usiErrPos,
		 );
		IF NOT xReadBusy THEN
			// allocate received module header
			stMDP_ModuleHeader	:= fbMDP_ReadModule.stMDP_ModuleHeader;
			// allocate information of startindexes in data buffer
			MEMCPY(ADR(arrStartIdx), ADR(fbMDP_ReadModule.arrStartIdx), SIZEOF(arrStartIdx) );
			// reset module content struct
			MEMSET( ADR(stMDP_ModuleContent), 0, SIZEOF(stMDP_ModuleContent) );
			// allocate received data to NIC struct
			stMDP_ModuleContent.uiLen		:= arrData[0];
			MEMCPY(ADR(stMDP_ModuleContent.udiProgMemAllocated),		ADR(arrData)+arrStartIdx[1],	MIN(arrStartIdx[2]-arrStartIdx[1],	SIZEOF(stMDP_ModuleContent.udiProgMemAllocated))     );
			MEMCPY(ADR(stMDP_ModuleContent.udiProgMemAvailable),		ADR(arrData)+arrStartIdx[2],	MIN(arrStartIdx[3]-arrStartIdx[2],	SIZEOF(stMDP_ModuleContent.udiProgMemAvailable))     );
//CE only	MEMCPY(ADR(stMDP_ModuleContent.udiStorageMemAllocated),		ADR(arrData)+arrStartIdx[3],	MIN(arrStartIdx[4]-arrStartIdx[3],	SIZEOF(stMDP_ModuleContent.udiStorageMemAllocated))     );
//CE omly	MEMCPY(ADR(stMDP_ModuleContent.udiStorageMemAvailable),		ADR(arrData)+arrStartIdx[4],	MIN(arrStartIdx[5]-arrStartIdx[4],	SIZEOF(stMDP_ModuleContent.udiStorageMemAvailable))     );
//CE only	MEMCPY(ADR(stMDP_ModuleContent.udiMemoryDivision),			ADR(arrData)+arrStartIdx[5],	MIN(arrStartIdx[6]-arrStartIdx[5],	SIZEOF(stMDP_ModuleContent.udiMemoryDivision))     );

			// reset FB
			xBusy 				:= FALSE;
		END_IF
	END_IF

	// check timeout
	TimeOut();
	IF TimeOut.Q THEN
		TimeOut(IN 				:= FALSE);
		xError					:= TRUE;
		udiErrID				:= INT_TO_UINT(eMDP_Err_PLC) * 16#10000 + INT_TO_UINT(eMDP_ErrPLC_TimeOut);
	END_IF
END_IF

IF xError THEN
	// reset FB
	xBusy 						:= FALSE;
END_IF

END_FUNCTION_BLOCK

// ---- POUs/MDP_Function_Blocks/FB_MDP_DiskMngmnt_ReadTBL1.TcPOU
FUNCTION_BLOCK FB_MDP_DiskMngmnt_ReadTBL1
VAR_INPUT
	xExecute			: BOOL;								// Function block execution is triggered by a rising edge at this input
	tTimeout			: TIME		:= DEFAULT_ADS_TIMEOUT;	// States the time before the function is cancelled
	usiModIdx			: USINT		:= 0;					// Index number of chosen MDP device
	sAmsNetId			: T_AmsNetId;						// keep empty '' for the local device	
END_VAR
VAR_OUTPUT
	xBusy				: BOOL;
	xError				: BOOL;
	udiErrID			: UDINT;
	usiErrPos			: USINT;							// If a subindex is not supported, iErrPos indicates at which subindex the error appears first
	stMDP_ModuleHeader	: ST_MDP_ModuleHeader;
	stMDP_ModuleContent	: ST_MDP_DiskMngmntTBL1;	
END_VAR
VAR
	fbMDP_ReadModule	: FB_MDP_ReadModule;
	arrData				: ARRAY[0..60] OF BYTE;			// requested data
	arrStartIdx			: ARRAY[0..20] OF UINT;			// startindexes in bytes of each subindex element

	stMDP_Addr			: ST_MDP_Addr;
	eModuleType			: E_MDP_ModuleType;
	usiSubIdxCount		: USINT;

	xSubExecute			: BOOL;
	xReadBusy			: BOOL;

	RisingEdge			: R_TRIG;
	TimeOut				: TON;								// general timeout
END_VAR

RisingEdge( CLK					:= xExecute );
IF NOT xBusy THEN											// FB only react to the external execute if it is not busy
	IF RisingEdge.Q THEN
		xBusy					:= TRUE;
		
		// reset variables
		xError					:= FALSE;
		udiErrID				:= 0;
		usiErrPos				:= 0;
		xSubExecute				:= TRUE;
	
		// specific values for NIC content
		stMDP_Addr.nArea		:= 16#08;
//		stMDP_Addr.nModuleId;								will be allocated dynamically
		stMDP_Addr.nTableId		:= 16#01;
//		stMDP_Addr.nFlag;									not used up to now
//		stMDP_Addr.nSubIdx;									all subindexes will be requested
		eModuleType				:= eMDP_ModT_DiskManagement;
		usiSubIdxCount			:= 7;						// TableId 16#01 contains 7 elements

		MEMSET( ADR(arrData), 0, SIZEOF(arrData) );			// reset buffer

		TimeOut(IN 				:= FALSE);
		TimeOut(PT 				:= tTimeout, IN := TRUE);
	END_IF
END_IF


IF xBusy THEN
	IF xSubExecute THEN
		xSubExecute 			:= FALSE;

		fbMDP_ReadModule( bExecute := FALSE );
		fbMDP_ReadModule(
			stMDP_Addr			:= stMDP_Addr,
			eModuleType			:= eModuleType,
			iModIdx				:= usiModIdx,
			iSubIdxCount		:= usiSubIdxCount,
			bExecute			:= TRUE,
			tTimeout			:= tTimeout,
			pDstBuf				:= ADR(arrData),
			cbDstBufLen			:= SIZEOF(arrData),
			sAmsNetId			:= sAmsNetId,

			bBusy				=> xReadBusy,
			bError				=> xError,
			nErrID				=> udiErrID,
			iErrPos				=> usiErrPos,
			stMDP_DynAddr		=> ,
			iModuleTypeCount	=> ,
			iModuleCount		=> ,
			stMDP_ModuleHeader	=> ,
			arrStartIdx			=> ,
		);
	ELSE
		fbMDP_ReadModule(
			bExecute			:= FALSE,

			bBusy				=> xReadBusy,
			bError				=> xError,
			nErrID 				=> udiErrID,
			iErrPos				=> usiErrPos,
		);
		IF NOT xReadBusy THEN
			// allocate received module header
			stMDP_ModuleHeader	:= fbMDP_ReadModule.stMDP_ModuleHeader;
			// allocate information of startindexes in data buffer
			MEMCPY(ADR(arrStartIdx), ADR(fbMDP_ReadModule.arrStartIdx), SIZEOF(arrStartIdx) );
			// reset module content struct
			MEMSET( ADR(stMDP_ModuleContent), 0, SIZEOF(stMDP_ModuleContent) );
			// allocate received data to DiskMngmntTBL1 struct
			stMDP_ModuleContent.uiLen		:= arrData[0];
			MEMCPY(ADR(stMDP_ModuleContent.sDriveLetter1), 	ADR(arrData)+arrStartIdx[1], MIN(arrStartIdx[2]-arrStartIdx[1], SIZEOF(stMDP_ModuleContent.sDriveLetter1)) );
			MEMCPY(ADR(stMDP_ModuleContent.sDriveLetter2), 	ADR(arrData)+arrStartIdx[2], MIN(arrStartIdx[3]-arrStartIdx[2], SIZEOF(stMDP_ModuleContent.sDriveLetter2))  );
			MEMCPY(ADR(stMDP_ModuleContent.sDriveLetter3), 	ADR(arrData)+arrStartIdx[3], MIN(arrStartIdx[4]-arrStartIdx[3], SIZEOF(stMDP_ModuleContent.sDriveLetter3)) );
			MEMCPY(ADR(stMDP_ModuleContent.sDriveLetter4), 	ADR(arrData)+arrStartIdx[4], MIN(arrStartIdx[5]-arrStartIdx[4], SIZEOF(stMDP_ModuleContent.sDriveLetter4)) );
			MEMCPY(ADR(stMDP_ModuleContent.sDriveLetter5),	ADR(arrData)+arrStartIdx[5], MIN(arrStartIdx[6]-arrStartIdx[5], SIZEOF(stMDP_ModuleContent.sDriveLetter5)) );
			MEMCPY(ADR(stMDP_ModuleContent.sDriveLetter6),	ADR(arrData)+arrStartIdx[6], MIN(arrStartIdx[7]-arrStartIdx[6], SIZEOF(stMDP_ModuleContent.sDriveLetter6)) );

			// reset FB
			xBusy 				:= FALSE;
		END_IF
	END_IF

	// check timeout
	TimeOut();
	IF TimeOut.Q THEN
		TimeOut(IN 				:= FALSE);
		xError					:= TRUE;
		udiErrID				:= INT_TO_UINT(eMDP_Err_PLC) * 16#10000 + INT_TO_UINT(eMDP_ErrPLC_TimeOut);
	END_IF
END_IF

IF xError THEN
	// reset FB
	xBusy 						:= FALSE;
END_IF

END_FUNCTION_BLOCK

// ---- POUs/MAIN.TcPOU
PROGRAM MAIN
//		8-2-2012
// 		This Program has been supplied by Beckhoff Automation As-Is and is intended only as an example 
//		implementation. Functionality is not guaranteed. 
//
VAR
	fb_InfoSafetyGroup1			: 	FB_InfoSafetyGroup ;
	fb_InfoConnection1			: 	FB_InfoConnectionIn ;
	fb_InfoConnection2			: 	FB_InfoConnectionOut ;
	fb_InfoAND					: 	FB_InfoAND ;
	fb_InfoEStop				: 	FB_InfoEStop ;
	fb_InfoAND2					: 	FB_InfoAND ;	
	fb_InfoTON					: 	FB_InfoTON ;
	fb_InfoTOF					: 	FB_InfoTOF ;	
	fb_InfoEDM					: 	FB_InfoEDM ;
	thgus: INT;
END_VAR

//		8-2-2012
// 		This Program has been supplied by Beckhoff Automation As-Is and is intended only as an example 
//		implementation. Functionality is not guaranteed. 
//
// Some standard I/O so EtherCAT BUS is running during TwinSAFE development
g_xOutput1 := 1 ;
g_xOutput2 := 1 ;
g_xOutput3 := 1 ;
g_xOutput4 := 1 ;

thgus;

IF g_bHMI_ScreenBeingDisplayed = 0 THEN
// Most Important Safety Project Info!!!
g_udiHMI_SerialNumber 				:= 		g_udiTS_SerialNumber ;
g_uiHMI_ProjectCRC 					:= 		g_uiTS_ProjectCRC ;

// Commands to TwinSAFE controller's safety  group
g_xTS_ErrAck 						:= 		g_xHMI_ErrAckPB ;
g_xTS_EStop_Reset 					:= 		g_xHMI_EStopResetPB ;

// Feedback from TwinSAFE controller's safety group
g_xHMI_SafetyGroup1_FBerrorLT 		:= 		g_xTS_SafetyGroup1_FBerror ;
g_xHMI_SafetyGroup1_COMerrorLT 		:= 		g_xTS_SafetyGroup1_COMerror ;

// Feedback from TwinSAFE controller's Function Blocks
g_xHMI_EDMerrorLT 					:= 		g_xTS_EDM_Error ;
g_xHMI_EStop_CompleteLT 			:= 		g_xTS_EStop_Complete ;
g_xHMI_EStop_errorLT 				:= 		g_xTS_EStop_Error ;
g_xHMI_EStop_OFF_Delay_CompleteLT 	:= 		g_xTS_EStop_OFF_Delay_Complete ;
g_xHMI_EStop_ON_Delay_CompleteLT 	:= 		g_xTS_EStop_ON_Delay_Complete ;

// TwinSAFE Group 1 Info
fb_InfoSafetyGroup1(
						stInfoData	:= 		g_stTS_InfoGroup1, 
						sState		=> 		g_sHMI_StatusGroup1 );

// TwinSAFE Connection 1 Info to EL1904 safety terminal
fb_InfoConnection1(
						stInfoData	:= 		g_stTS_InfoConnection1, 
						sState		=> 		g_sHMI_StateConn1, 
						sDiag		=> 		g_sHMI_DiagConn1, 
						xChannel1	=> 		g_xHMI_EL1904Ch1, 
						xChannel2	=> 		g_xHMI_EL1904Ch2, 
						xChannel3	=> 		g_xHMI_EL1904Ch3, 
						xChannel4	=> 		g_xHMI_EL1904Ch4 );
	
// TwinSAFE Connection 2 Info to EL2904 safety terminal
fb_InfoConnection2(
						stInfoData	:= 		g_stTS_InfoConnection2, 
						sState		=> 		g_sHMI_StateConn2, 
						sDiag		=> 		g_sHMI_DiagConn2, 
						xChannel1	=> 		g_xHMI_EL2904Ch1, 
						xChannel2	=> 		g_xHMI_EL2904Ch2, 
						xChannel3	=> 		g_xHMI_EL2904Ch3, 
						xChannel4	=> 		g_xHMI_EL2904Ch4 );	
								
// TwinSAFE First AND safety FB Info
fb_InfoAND(				stInfoData	:= 		g_stTS_InfoAND1, 
						sState		=> 		g_sHMI_StatusAND1 );

// TwinSAFE ESTOP safety FB Info
fb_InfoEStop(			stInfoData	:= 		g_stTS_InfoEStop1, 
						sState		=> 		g_sHMI_StatusEStop1, 		
						sDiag		=> 		g_sHMI_DiagEStop1 );

// TwinSAFE Second AND safety FB Info
fb_InfoAND2(			stInfoData	:= 		g_stTS_InfoAND2, 
						sState		=> 		g_sHMI_StatusAND2 );
						
// TwinSAFE TON safety FB Info
fb_InfoTON(				stInfoData	:= 		g_stTS_InfoTON, 
						sState		=> 		g_sHMI_StatusTON );

// TwinSAFE TOF safety FB Info
fb_InfoTOF(				stInfoData	:= 		g_stTS_InfoTOF, 
						sState		=> 		g_sHMI_StatusTOF );

// TwinSAFE EDM safety FB Info
fb_InfoEDM(				stInfoData	:= 		g_stTS_InfoEDM, 
						sState		=> 		g_sHMI_StatusEDM, 
						sDiag		=> 		g_sHMI_DiagEDM );	
END_IF ;

// Get Control System Diagnostics 
EtherCAT_Diag() ;
System_Functions() ;

//  ***********************************************************************
//	*																	  *
//  * NEVER try to WRITE to a safety terminal's CoE area (only read)!!!!  *
//	*																	  *
//	***********************************************************************			
						
// Get additional diagnostic info from the EL6900 saftey logic terminal
EL6900_ADS_Reads() ;

// Get additional diagnostic info from the EL1904 saftey terminal
EL1904_ADS_Reads() ;					

// Get additional diagnostic info from the EP1908-0002 saftey module
//EP1908_ADS_Reads() ;

// Get additional diagnostic info from the EL1904 saftey terminal
EL2904_ADS_Reads() ;

// Get additional diagnostic info from the EL6930 saftey logic terminal
//EL6930_ADS_Reads() ;

// Get additional diagnostic info from the AX5805 Safe Motion Module 
//AX5805_ADS_Reads() ;

END_PROGRAM

// ---- POUs/TwinSAFE_Function_Blocks_Info/FB_InfoSafetyGroup.TcPOU
FUNCTION_BLOCK FB_InfoSafetyGroup
VAR_INPUT
	stInfoData 		: 		DUT_ST_InfoData ;
END_VAR
VAR_OUTPUT
	sState 			: 		STRING ;
END_VAR
VAR
END_VAR

// Safety Group State

// Value 1 - RUN: All function blocks and TwinSAFE connections assigned to the TwinSAFE
// group operate properly, and all TwinSAFE connections assigned to the TwinSAFE 
// group are up and running
IF stInfoData.usiMapState 		= 	1 THEN
				sState 			:= 	'RUN - All FBs and Connections Operating Properly' ;

// Value 2 - Stop: The state TwinSAFE goes to after initialization
ELSIF stInfoData.usiMapState 	= 	2 THEN
				sState 			:= 	'STOP - State After Initialization' ;

// Value 3 - SAFE: All function blocks and TwinSAFE connections assigned to the TwinSAFE
// group operate properly, and at least one of the TwinSAFE connections
// assigned to the TwinSAFE group is not up and running
ELSIF stInfoData.usiMapState 	= 	3 THEN
				sState 			:= 	'SAFE - An Assigned Connection Not Up and Running' ;

// Value 4 - ERROR: At least one assigned function block or one assigned TwinSAFE connection
// has reported an error 
ELSIF stInfoData.usiMapState 	= 	4 THEN
				sState 			:= 	'ERROR - FB or Connection in Error State' ;

// Value 5 - RESET: A positive edge (FALSE -> TRUE) for the safety group error Ack
// of a function block or a TwinSAFE connection error was detected on the ERR_ACK input.
// The system is waiting for a negative edge of the ERR_ACK input.
ELSIF stInfoData.usiMapState 	= 	5 THEN
				sState 			:= 	'RESET - ErrAck TRUE, Waiting For ErrAck FALSE' ;

// Value 0: Safety group does not exist or safety controller has not been started
ELSE
				sState 			:= 	'Unknown' ;
END_IF

// The Safety Group Has No Diagnostic Byte to Decode

END_FUNCTION_BLOCK

// ---- POUs/TwinSAFE_Function_Blocks_Info/FB_InfoEStop.TcPOU
FUNCTION_BLOCK FB_InfoEStop
VAR_INPUT
	stInfoData 			:		DUT_ST_InfoDataFB ;
END_VAR
VAR_OUTPUT
	sState 				: 		STRING ;
	sDiag 				: 		STRING ;
	END_VAR
VAR
END_VAR

// EStop FB's State
IF stInfoData.usiMapState 			= 	0 THEN
				sState 				:= 	'Undefined' ;
	ELSIF stInfoData.usiMapState 	= 	1 THEN
				sState 				:= 	'RUN' ;
	ELSIF stInfoData.usiMapState	=	2 THEN
				sState 				:= 'STOP' ;
	ELSIF stInfoData.usiMapState 	= 	3 THEN
				sState 				:= 	'SAFE' ;
	ELSIF stInfoData.usiMapState 	= 	4 THEN
				sState 				:= 	'ERROR' ;
	ELSIF stInfoData.usiMapState 	= 	5 THEN
				sState 				:= 	'RESET' ;
	ELSIF stInfoData.usiMapState 	= 	6 THEN
				sState 				:= 	'START' ;
	ELSIF stInfoData.usiMapState 	= 	8 THEN
				sState 				:= 	'DELAYOUT' ;
	ELSE
				sState 				:= 	'Unknown' ;
END_IF

// EStop FB's Diagnostics
IF stInfoData.uiMapDiag 			= 	0 THEN
				sDiag 				:= 	'No Error' ;
	ELSIF stInfoData.uiMapDiag		= 	1 THEN
				sDiag 				:= 	'Discrepancy Error Input Group 1' ;
	ELSIF stInfoData.uiMapDiag 		= 	2 THEN
				sDiag 				:= 	'Discrepancy Error Input Group 2' ;
	ELSIF stInfoData.uiMapDiag 		= 	4 THEN
				sDiag 				:= 	'Discrepancy Error Input Group 3' ;
	ELSIF stInfoData.uiMapDiag 		= 	8 THEN
				sDiag 				:= 	'Discrepancy Error Input Group 4' ;
	ELSIF stInfoData.uiMapDiag 		= 	16 THEN
				sDiag 				:= 	'EDM 1 Monitoring Error' ;	
	ELSIF stInfoData.uiMapDiag 		= 	32 THEN
				sDiag 				:= 	'EDM 2 Monitoring Error' ;	
	ELSE
				sDiag 				:= 	'Unknown' ;
END_IF

END_FUNCTION_BLOCK

// ---- POUs/TwinSAFE_Function_Blocks_Info/FB_InfoTOF.TcPOU
FUNCTION_BLOCK FB_InfoTOF
VAR_INPUT
	stInfoData 		: 		DUT_ST_InfoDataFB ;
END_VAR
VAR_OUTPUT
	sState 			: 		STRING ;
END_VAR
VAR
END_VAR

// Timer-OFF (TOF) FB's State
IF stInfoData.usiMapState 			= 	0 THEN
				sState 				:= 	'Undefined' ;
	ELSIF stInfoData.usiMapState 	= 	1 THEN
				sState 				:= 	'RUN' ;
	ELSIF stInfoData.usiMapState 	= 	2 THEN
				sState 				:= 	'STOP' ;
	ELSIF stInfoData.usiMapState 	= 	3 THEN
				sState 				:= 	'SAFE' ;
	ELSIF stInfoData.usiMapState 	= 	8 THEN
				sState 				:= 	'DelayOut' ;
	ELSE
				sState 				:= 	'Unknown' ;
END_IF

// The Timer-OFF (TOF) FB Has No Diagnostic Byte to Decode

END_FUNCTION_BLOCK

// ---- POUs/MDP_Function_Blocks/FB_MDP_DiskMngmnt_ReadTBL2.TcPOU
FUNCTION_BLOCK FB_MDP_DiskMngmnt_ReadTBL2
VAR_INPUT
	xExecute			: BOOL;								// Function block execution is triggered by a rising edge at this input
	tTimeout			: TIME		:= DEFAULT_ADS_TIMEOUT;	// States the time before the function is cancelled
	usiModIdx			: USINT		:= 0;					// Index number of chosen MDP device
	sAmsNetId			: T_AmsNetId;						// keep empty '' for the local device	
END_VAR
VAR_OUTPUT
	xBusy				: BOOL;
	xError				: BOOL;
	udiErrID			: UDINT;
	usiErrPos			: USINT;							// If a subindex is not supported, iErrPos indicates at which subindex the error appears first
	stMDP_ModuleHeader	: ST_MDP_ModuleHeader;
	stMDP_ModuleContent	: ST_MDP_DiskMngmntTBL2;	
END_VAR
VAR
	fbMDP_ReadModule	: FB_MDP_ReadModule;
	arrData				: ARRAY[0..799] OF BYTE;			// requested data
	arrStartIdx			: ARRAY[0..255] OF UINT;			// startindexes in bytes of each subindex element

	stMDP_Addr			: ST_MDP_Addr;
	eModuleType			: E_MDP_ModuleType;
	usiSubIdxCount		: USINT;

	xSubExecute			: BOOL;
	xReadBusy			: BOOL;

	RisingEdge			: R_TRIG;
	TimeOut				: TON;								// general timeout
END_VAR

RisingEdge( CLK					:= xExecute );
IF NOT xBusy THEN											// FB only react to the external execute if it is not busy
	IF RisingEdge.Q THEN
		xBusy					:= TRUE;
		
		// reset variables
		xError					:= FALSE;
		udiErrID				:= 0;
		usiErrPos				:= 0;
		xSubExecute				:= TRUE;
	
		// specific values for NIC content
		stMDP_Addr.nArea		:= 16#08;
//		stMDP_Addr.nModuleId;								will be allocated dynamically
		stMDP_Addr.nTableId		:= 16#01;
//		stMDP_Addr.nFlag;									not used up to now
//		stMDP_Addr.nSubIdx;									all subindexes will be requested
		eModuleType				:= eMDP_ModT_NIC;
		usiSubIdxCount			:= 7;						// TableId 16#01 contains 6 elements

		MEMSET( ADR(arrData), 0, SIZEOF(arrData) );			// reset buffer

		TimeOut(IN 				:= FALSE);
		TimeOut(PT 				:= tTimeout, IN := TRUE);
	END_IF
END_IF


IF xBusy THEN
	IF xSubExecute THEN
		xSubExecute 			:= FALSE;

		fbMDP_ReadModule( bExecute := FALSE );
		fbMDP_ReadModule(
			stMDP_Addr			:= stMDP_Addr,
			eModuleType			:= eModuleType,
			iModIdx				:= usiModIdx,
			iSubIdxCount		:= usiSubIdxCount,
			bExecute			:= TRUE,
			tTimeout			:= tTimeout,
			pDstBuf				:= ADR(arrData),
			cbDstBufLen			:= SIZEOF(arrData),
			sAmsNetId			:= sAmsNetId,

			bBusy				=> xReadBusy,
			bError				=> xError,
			nErrID				=> udiErrID,
			iErrPos				=> usiErrPos,
			stMDP_DynAddr		=> ,
			iModuleTypeCount	=> ,
			iModuleCount		=> ,
			stMDP_ModuleHeader	=> ,
			arrStartIdx			=> ,
		);
	ELSE
		fbMDP_ReadModule(
			bExecute			:= FALSE,

			bBusy				=> xReadBusy,
			bError				=> xError,
			nErrID 				=> udiErrID,
			iErrPos				=> usiErrPos,
		);
		IF NOT xReadBusy THEN
			// allocate received module header
			stMDP_ModuleHeader	:= fbMDP_ReadModule.stMDP_ModuleHeader;
			// allocate information of startindexes in data buffer
			MEMCPY(ADR(arrStartIdx), ADR(fbMDP_ReadModule.arrStartIdx), SIZEOF(arrStartIdx) );
			// reset module content struct
			MEMSET( ADR(stMDP_ModuleContent), 0, SIZEOF(stMDP_ModuleContent) );
			// allocate received data to DiskMngmntTBL2 struct
			stMDP_ModuleContent.uiLen		:= arrData[0];
			MEMCPY(ADR(stMDP_ModuleContent.sVolumeLabel1), 	ADR(arrData)+arrStartIdx[1], MIN(arrStartIdx[2]-arrStartIdx[1], SIZEOF(stMDP_ModuleContent.sVolumeLabel1)) );
			MEMCPY(ADR(stMDP_ModuleContent.sVolumeLabel2), 	ADR(arrData)+arrStartIdx[2], MIN(arrStartIdx[3]-arrStartIdx[2], SIZEOF(stMDP_ModuleContent.sVolumeLabel2))  );
			MEMCPY(ADR(stMDP_ModuleContent.sVolumeLabel3), 	ADR(arrData)+arrStartIdx[3], MIN(arrStartIdx[4]-arrStartIdx[3], SIZEOF(stMDP_ModuleContent.sVolumeLabel3)) );
			MEMCPY(ADR(stMDP_ModuleContent.sVolumeLabel4), 	ADR(arrData)+arrStartIdx[4], MIN(arrStartIdx[5]-arrStartIdx[4], SIZEOF(stMDP_ModuleContent.sVolumeLabel4)) );
			MEMCPY(ADR(stMDP_ModuleContent.sVolumeLabel5),	ADR(arrData)+arrStartIdx[5], MIN(arrStartIdx[6]-arrStartIdx[5], SIZEOF(stMDP_ModuleContent.sVolumeLabel5)) );
			MEMCPY(ADR(stMDP_ModuleContent.sVolumeLabel6),	ADR(arrData)+arrStartIdx[6], MIN(arrStartIdx[7]-arrStartIdx[6], SIZEOF(stMDP_ModuleContent.sVolumeLabel6)) );

			// reset FB
			xBusy 				:= FALSE;
		END_IF
	END_IF

	// check timeout
	TimeOut();
	IF TimeOut.Q THEN
		TimeOut(IN 				:= FALSE);
		xError					:= TRUE;
		udiErrID				:= INT_TO_UINT(eMDP_Err_PLC) * 16#10000 + INT_TO_UINT(eMDP_ErrPLC_TimeOut);
	END_IF
END_IF

IF xError THEN
	// reset FB
	xBusy 						:= FALSE;
END_IF

END_FUNCTION_BLOCK

// ---- POUs/MDP_Function_Blocks/FB_MDP_DiskMngmnt_ReadTBL3.TcPOU
FUNCTION_BLOCK FB_MDP_DiskMngmnt_ReadTBL3
VAR_INPUT
	xExecute			: BOOL;								// Function block execution is triggered by a rising edge at this input
	tTimeout			: TIME		:= DEFAULT_ADS_TIMEOUT;	// States the time before the function is cancelled
	usiModIdx			: USINT		:= 0;					// Index number of chosen MDP device
	sAmsNetId			: T_AmsNetId;						// keep empty '' for the local device	
END_VAR
VAR_OUTPUT
	xBusy				: BOOL;
	xError				: BOOL;
	udiErrID			: UDINT;
	usiErrPos			: USINT;							// If a subindex is not supported, iErrPos indicates at which subindex the error appears first
	stMDP_ModuleHeader	: ST_MDP_ModuleHeader;
	stMDP_ModuleContent	: ST_MDP_DiskMngmntTBL3;	
END_VAR
VAR
	fbMDP_ReadModule	: FB_MDP_ReadModule;
	arrData				: ARRAY[0..799] OF BYTE;			// requested data
	arrStartIdx			: ARRAY[0..255] OF UINT;			// startindexes in bytes of each subindex element

	stMDP_Addr			: ST_MDP_Addr;
	eModuleType			: E_MDP_ModuleType;
	usiSubIdxCount		: USINT;

	xSubExecute			: BOOL;
	xReadBusy			: BOOL;

	RisingEdge			: R_TRIG;
	TimeOut				: TON;								// general timeout
END_VAR

RisingEdge( CLK					:= xExecute );
IF NOT xBusy THEN											// FB only react to the external execute if it is not busy
	IF RisingEdge.Q THEN
		xBusy					:= TRUE;
		
		// reset variables
		xError					:= FALSE;
		udiErrID				:= 0;
		usiErrPos				:= 0;
		xSubExecute				:= TRUE;
	
		// specific values for NIC content
		stMDP_Addr.nArea		:= 16#08;
//		stMDP_Addr.nModuleId;								will be allocated dynamically
		stMDP_Addr.nTableId		:= 16#01;
//		stMDP_Addr.nFlag;									not used up to now
//		stMDP_Addr.nSubIdx;									all subindexes will be requested
		eModuleType				:= eMDP_ModT_NIC;
		usiSubIdxCount			:= 7;						// TableId 16#01 contains 6 elements

		MEMSET( ADR(arrData), 0, SIZEOF(arrData) );			// reset buffer

		TimeOut(IN 				:= FALSE);
		TimeOut(PT 				:= tTimeout, IN := TRUE);
	END_IF
END_IF


IF xBusy THEN
	IF xSubExecute THEN
		xSubExecute 			:= FALSE;

		fbMDP_ReadModule( bExecute := FALSE );
		fbMDP_ReadModule(
			stMDP_Addr			:= stMDP_Addr,
			eModuleType			:= eModuleType,
			iModIdx				:= usiModIdx,
			iSubIdxCount		:= usiSubIdxCount,
			bExecute			:= TRUE,
			tTimeout			:= tTimeout,
			pDstBuf				:= ADR(arrData),
			cbDstBufLen			:= SIZEOF(arrData),
			sAmsNetId			:= sAmsNetId,

			bBusy				=> xReadBusy,
			bError				=> xError,
			nErrID				=> udiErrID,
			iErrPos				=> usiErrPos,
			stMDP_DynAddr		=> ,
			iModuleTypeCount	=> ,
			iModuleCount		=> ,
			stMDP_ModuleHeader	=> ,
			arrStartIdx			=> ,
		);
	ELSE
		fbMDP_ReadModule(
			bExecute			:= FALSE,

			bBusy				=> xReadBusy,
			bError				=> xError,
			nErrID 				=> udiErrID,
			iErrPos				=> usiErrPos,
		);
		IF NOT xReadBusy THEN
			// allocate received module header
			stMDP_ModuleHeader	:= fbMDP_ReadModule.stMDP_ModuleHeader;
			// allocate information of startindexes in data buffer
			MEMCPY(ADR(arrStartIdx), ADR(fbMDP_ReadModule.arrStartIdx), SIZEOF(arrStartIdx) );
			// reset module content struct
			MEMSET( ADR(stMDP_ModuleContent), 0, SIZEOF(stMDP_ModuleContent) );
			// allocate received data to DiskMngmntTBL3 struct
			stMDP_ModuleContent.uiLen		:= arrData[0];
			MEMCPY(ADR(stMDP_ModuleContent.sFileSystemName1), 	ADR(arrData)+arrStartIdx[1], MIN(arrStartIdx[2]-arrStartIdx[1], SIZEOF(stMDP_ModuleContent.sFileSystemName1)) );
			MEMCPY(ADR(stMDP_ModuleContent.sFileSystemName2), 	ADR(arrData)+arrStartIdx[2], MIN(arrStartIdx[3]-arrStartIdx[2], SIZEOF(stMDP_ModuleContent.sFileSystemName2))  );
			MEMCPY(ADR(stMDP_ModuleContent.sFileSystemName3), 	ADR(arrData)+arrStartIdx[3], MIN(arrStartIdx[4]-arrStartIdx[3], SIZEOF(stMDP_ModuleContent.sFileSystemName3)) );
			MEMCPY(ADR(stMDP_ModuleContent.sFileSystemName4), 	ADR(arrData)+arrStartIdx[4], MIN(arrStartIdx[5]-arrStartIdx[4], SIZEOF(stMDP_ModuleContent.sFileSystemName4)) );
			MEMCPY(ADR(stMDP_ModuleContent.sFileSystemName5),	ADR(arrData)+arrStartIdx[5], MIN(arrStartIdx[6]-arrStartIdx[5], SIZEOF(stMDP_ModuleContent.sFileSystemName5)) );
			MEMCPY(ADR(stMDP_ModuleContent.sFileSystemName6),	ADR(arrData)+arrStartIdx[6], MIN(arrStartIdx[7]-arrStartIdx[6], SIZEOF(stMDP_ModuleContent.sFileSystemName6)) );

			// reset FB
			xBusy 				:= FALSE;
		END_IF
	END_IF

	// check timeout
	TimeOut();
	IF TimeOut.Q THEN
		TimeOut(IN 				:= FALSE);
		xError					:= TRUE;
		udiErrID				:= INT_TO_UINT(eMDP_Err_PLC) * 16#10000 + INT_TO_UINT(eMDP_ErrPLC_TimeOut);
	END_IF
END_IF

IF xError THEN
	// reset FB
	xBusy 						:= FALSE;
END_IF

END_FUNCTION_BLOCK

// ---- POUs/MDP_Function_Blocks/FB_MDP_DiskMngmnt_ReadTBL4.TcPOU
FUNCTION_BLOCK FB_MDP_DiskMngmnt_ReadTBL4
VAR_INPUT
	xExecute			: BOOL;								// Function block execution is triggered by a rising edge at this input
	tTimeout			: TIME		:= DEFAULT_ADS_TIMEOUT;	// States the time before the function is cancelled
	usiModIdx			: USINT		:= 0;					// Index number of chosen MDP device
	sAmsNetId			: T_AmsNetId;						// keep empty '' for the local device	
END_VAR
VAR_OUTPUT
	xBusy				: BOOL;
	xError				: BOOL;
	udiErrID			: UDINT;
	usiErrPos			: USINT;							// If a subindex is not supported, iErrPos indicates at which subindex the error appears first
	stMDP_ModuleHeader	: ST_MDP_ModuleHeader;
	stMDP_ModuleContent	: ST_MDP_DiskMngmntTBL4;	
END_VAR
VAR
	fbMDP_ReadModule	: FB_MDP_ReadModule;
	arrData				: ARRAY[0..799] OF BYTE;			// requested data
	arrStartIdx			: ARRAY[0..255] OF UINT;			// startindexes in bytes of each subindex element

	stMDP_Addr			: ST_MDP_Addr;
	eModuleType			: E_MDP_ModuleType;
	usiSubIdxCount		: USINT;

	xSubExecute			: BOOL;
	xReadBusy			: BOOL;

	RisingEdge			: R_TRIG;
	TimeOut				: TON;								// general timeout
END_VAR

RisingEdge( CLK					:= xExecute );
IF NOT xBusy THEN											// FB only react to the external execute if it is not busy
	IF RisingEdge.Q THEN
		xBusy					:= TRUE;
		
		// reset variables
		xError					:= FALSE;
		udiErrID				:= 0;
		usiErrPos				:= 0;
		xSubExecute				:= TRUE;
	
		// specific values for NIC content
		stMDP_Addr.nArea		:= 16#08;
//		stMDP_Addr.nModuleId;								will be allocated dynamically
		stMDP_Addr.nTableId		:= 16#01;
//		stMDP_Addr.nFlag;									not used up to now
//		stMDP_Addr.nSubIdx;									all subindexes will be requested
		eModuleType				:= eMDP_ModT_NIC;
		usiSubIdxCount			:= 7;						// TableId 16#01 contains 6 elements

		MEMSET( ADR(arrData), 0, SIZEOF(arrData) );			// reset buffer

		TimeOut(IN 				:= FALSE);
		TimeOut(PT 				:= tTimeout, IN := TRUE);
	END_IF
END_IF


IF xBusy THEN
	IF xSubExecute THEN
		xSubExecute 			:= FALSE;

		fbMDP_ReadModule( bExecute := FALSE );
		fbMDP_ReadModule(
			stMDP_Addr			:= stMDP_Addr,
			eModuleType			:= eModuleType,
			iModIdx				:= usiModIdx,
			iSubIdxCount		:= usiSubIdxCount,
			bExecute			:= TRUE,
			tTimeout			:= tTimeout,
			pDstBuf				:= ADR(arrData),
			cbDstBufLen			:= SIZEOF(arrData),
			sAmsNetId			:= sAmsNetId,

